TYPE "READ_AXES_POSITIONS_CH"
// stored: IsFailsafeCompliant false
   STRUCT
      READING_FAULT_1 : Bool;   // READING FAULT 1
      READING_DONE_1 : Bool;   // READING DONE 1
      REQUEST_1 : Bool;   // REQUEST 1
      READING_FAULT_2 : Bool;   // READING FAULT 2
      READING_DONE_2 : Bool;   // READING DONE 2
      REQUEST_2 : Bool;   // REQUEST 2
      READING_FAULT_3 : Bool;   // READING FAULT 3
      READING_DONE_3 : Bool;   // READING DONE 3
      REQUEST_3 : Bool;   // REQUEST 3
      FAULT_1 : Bool;   // FAULT 1
      FAULT_2 : Bool;   // FAULT 2
      FAULT_3 : Bool;   // FAULT 3
      IS : Bool;   // INMEDIATE STOP ALARMS / IMMEDIATE STOP ALARMS
      IS_SEOC : Bool;   // INMEDIATE STOP & STOP END OF CYCLE ALARMS / IMMEDIATE STOP & STOP END OF CYCLE ALARMS
      RHP : Bool;   // RETURN HOME POSITION ALARMS
      RHP_SEOC : Bool;   // RETURN HOME POSITION & STOP END OF CYCLE ALARMS
      SEOC : Bool;   // STOP END OF CYCLE ALARMS
      IS_WARNING : Bool;   // INMEDIATE STOP WARNING / IMMEDIATE STOP WARNING
      RHP_WARNING : Bool;   // RETURN HOME POSITION WARNING
      SEOC_WARNING : Bool;   // STOP END OF CYCLE WARNING
      WARNINGS : Bool;   // WARNINGS
      Help : Bool;   // Help
      Aux : Bool;   // Aux
      Aux1 : Bool;   // Aux1
      Aux2 : Bool;   // Aux2
      Aux3 : Bool;   // Aux3
      Aux4 : Bool;   // Aux4
      Aux5 : Bool;   // Aux5
      Aux6 : Bool;   // Aux6
      Aux7 : Bool;   // Aux7
      READING_STATUS : Word;   // READING STATUS
      POSITION_AXIS_1 : DWord;   // POSITION AXIS 1
      POSITION_AXIS_2 : DWord;   // POSITION AXIS 2
      POSITION_AXIS_3 : DWord;   // POSITION AXIS 3
      POSITION_AXIS_4 : DWord;   // POSITION AXIS 4
      POSITION_AXIS_5 : DWord;   // POSITION AXIS 5
      POSITION_AXIS_6 : DWord;   // POSITION AXIS 6
      POSITION_AXIS_7 : DWord;   // POSITION AXIS 7
      POSITION_AXIS_8 : DWord;   // POSITION AXIS 8
      POSITION_AXIS_9 : DWord;   // POSITION AXIS 9
      POSITION_AXIS_10 : DWord;   // POSITION AXIS 10
      POSITION_AXIS_11 : DWord;   // POSITION AXIS 11
      POSITION_AXIS_12 : DWord;   // POSITION AXIS 12
      POSITION_AXIS_13 : DWord;   // POSITION AXIS 13
      POSITION_AXIS_14 : DWord;   // POSITION AXIS 14
      POSITION_AXIS_15 : DWord;   // POSITION AXIS 15
      POSITION_AXIS_16 : DWord;   // POSITION AXIS 16
      POSITION_AXIS_17 : DWord;   // POSITION AXIS 17
      POSITION_AXIS_18 : DWord;   // POSITION AXIS 18
      POSITION_AXIS_19 : DWord;   // POSITION AXIS 19
      POSITION_AXIS_20 : DWord;   // POSITION AXIS 20
      CH_Reading_1 : Struct   // CH Reading 1
         SYNTAX_ID : Byte := BYTE#16#82;   // SYNTAX ID
         Area_Unit : Byte := BYTE#16#41;   // Area_Unit
         Column : Word := WORD#16#0002;   // Column
         Line : Word := WORD#16#0001;   // Line
         BlockType : Byte := BYTE#16#74;   // Block Type
         NumOfLine : Byte := BYTE#16#01;   // Number Of Line
         DataType : Byte := BYTE#16#0F;   // Data Type
         Length : Byte := BYTE#16#08;   // Length
      END_STRUCT;
      CH_Reading_2 : Struct   // CH Reading 2
         SYNTAX_ID : Byte := BYTE#16#82;   // SYNTAX ID
         Area_Unit : Byte := BYTE#16#41;   // Area_Unit
         Column : Word := WORD#16#0002;   // Column
         Line : Word := WORD#16#0002;   // Line
         BlockType : Byte := BYTE#16#74;   // Block Type
         NumOfLine : Byte := BYTE#16#01;   // Number Of Line
         DataType : Byte := BYTE#16#0F;   // Data Type
         Length : Byte := BYTE#16#08;   // Length
      END_STRUCT;
      CH_Reading_3 : Struct   // CH Reading 3
         SYNTAX_ID : Byte := BYTE#16#82;   // SYNTAX ID
         Area_Unit : Byte := BYTE#16#41;   // Area_Unit
         Column : Word := WORD#16#0002;   // Column
         Line : Word := WORD#16#0003;   // Line
         BlockType : Byte := BYTE#16#74;   // Block Type
         NumOfLine : Byte := BYTE#16#01;   // Number Of Line
         DataType : Byte := BYTE#16#0F;   // Data Type
         Length : Byte := BYTE#16#08;   // Length
      END_STRUCT;
      CH_Reading_4 : Struct   // CH Reading 4
         SYNTAX_ID : Byte := BYTE#16#82;   // SYNTAX ID
         Area_Unit : Byte := BYTE#16#41;   // Area_Unit
         Column : Word := WORD#16#0002;   // Column
         Line : Word := WORD#16#0004;   // Line
         BlockType : Byte := BYTE#16#74;   // Block Type
         NumOfLine : Byte := BYTE#16#01;   // Number Of Line
         DataType : Byte := BYTE#16#0F;   // Data Type
         Length : Byte := BYTE#16#08;   // Length
      END_STRUCT;
      CH_Reading_5 : Struct   // CH Reading 5
         SYNTAX_ID : Byte := BYTE#16#82;   // SYNTAX ID
         Area_Unit : Byte := BYTE#16#41;   // Area_Unit
         Column : Word := WORD#16#0002;   // Column
         Line : Word := WORD#16#0005;   // Line
         BlockType : Byte := BYTE#16#74;   // Block Type
         NumOfLine : Byte := BYTE#16#01;   // Number Of Line
         DataType : Byte := BYTE#16#0F;   // Data Type
         Length : Byte := BYTE#16#08;   // Length
      END_STRUCT;
      CH_Reading_6 : Struct   // CH Reading 6
         SYNTAX_ID : Byte := BYTE#16#82;   // SYNTAX ID
         Area_Unit : Byte := BYTE#16#41;   // Area_Unit
         Column : Word := WORD#16#0002;   // Column
         Line : Word := WORD#16#0006;   // Line
         BlockType : Byte := BYTE#16#74;   // Block Type
         NumOfLine : Byte := BYTE#16#01;   // Number Of Line
         DataType : Byte := BYTE#16#0F;   // Data Type
         Length : Byte := BYTE#16#08;   // Length
      END_STRUCT;
      CH_Reading_7 : Struct   // CH Reading 7
         SYNTAX_ID : Byte := BYTE#16#82;   // SYNTAX ID
         Area_Unit : Byte := BYTE#16#41;   // Area_Unit
         Column : Word := WORD#16#0002;   // Column
         Line : Word := WORD#16#0007;   // Line
         BlockType : Byte := BYTE#16#74;   // Block Type
         NumOfLine : Byte := BYTE#16#01;   // Number Of Line
         DataType : Byte := BYTE#16#0F;   // Data Type
         Length : Byte := BYTE#16#08;   // Length
      END_STRUCT;
      CH_Reading_8 : Struct   // CH Reading 8
         SYNTAX_ID : Byte := BYTE#16#82;   // SYNTAX ID
         Area_Unit : Byte := BYTE#16#41;   // Area_Unit
         Column : Word := WORD#16#0002;   // Column
         Line : Word := WORD#16#0008;   // Line
         BlockType : Byte := BYTE#16#74;   // Block Type
         NumOfLine : Byte := BYTE#16#01;   // Number Of Line
         DataType : Byte := BYTE#16#0F;   // Data Type
         Length : Byte := BYTE#16#08;   // Length
      END_STRUCT;
      CH_Reading_9 : Struct   // CH Reading 9
         SYNTAX_ID : Byte := BYTE#16#82;   // SYNTAX ID
         Area_Unit : Byte := BYTE#16#41;   // Area_Unit
         Column : Word := WORD#16#0002;   // Column
         Line : Word := WORD#16#0009;   // Line
         BlockType : Byte := BYTE#16#74;   // Block Type
         NumOfLine : Byte := BYTE#16#01;   // Number Of Line
         DataType : Byte := BYTE#16#0F;   // Data Type
         Length : Byte := BYTE#16#08;   // Length
      END_STRUCT;
      CH_Reading_10 : Struct   // CH Reading 10
         SYNTAX_ID : Byte := BYTE#16#82;   // SYNTAX ID
         Area_Unit : Byte := BYTE#16#41;   // Area_Unit
         Column : Word := WORD#16#0002;   // Column
         Line : Word := WORD#16#000A;   // Line
         BlockType : Byte := BYTE#16#73;   // Block Type
         NumOfLine : Byte := BYTE#16#01;   // Number Of Line
         DataType : Byte := BYTE#16#0F;   // Data Type
         Length : Byte := BYTE#16#08;   // Length
      END_STRUCT;
      CH_Reading_11 : Struct   // CH Reading 11
         SYNTAX_ID : Byte := BYTE#16#82;   // SYNTAX ID
         Area_Unit : Byte := BYTE#16#41;   // Area_Unit
         Column : Word := WORD#16#0002;   // Column
         Line : Word := WORD#16#000B;   // Line
         BlockType : Byte := BYTE#16#74;   // Block Type
         NumOfLine : Byte := BYTE#16#01;   // Number Of Line
         DataType : Byte := BYTE#16#0F;   // Data Type
         Length : Byte := BYTE#16#08;   // Length
      END_STRUCT;
      CH_Reading_12 : Struct   // CH Reading 12
         SYNTAX_ID : Byte := BYTE#16#82;   // SYNTAX ID
         Area_Unit : Byte := BYTE#16#41;   // Area_Unit
         Column : Word := WORD#16#0002;   // Column
         Line : Word := WORD#16#000C;   // Line
         BlockType : Byte := BYTE#16#74;   // Block Type
         NumOfLine : Byte := BYTE#16#01;   // Number Of Line
         DataType : Byte := BYTE#16#0F;   // Data Type
         Length : Byte := BYTE#16#08;   // Length
      END_STRUCT;
      CH_Reading_13 : Struct   // CH Reading 13
         SYNTAX_ID : Byte := BYTE#16#82;   // SYNTAX ID
         Area_Unit : Byte := BYTE#16#41;   // Area_Unit
         Column : Word := WORD#16#0002;   // Column
         Line : Word := WORD#16#000D;   // Line
         BlockType : Byte := BYTE#16#74;   // Block Type
         NumOfLine : Byte := BYTE#16#01;   // Number Of Line
         DataType : Byte := BYTE#16#0F;   // Data Type
         Length : Byte := BYTE#16#08;   // Length
      END_STRUCT;
      CH_Reading_14 : Struct   // CH Reading 14
         SYNTAX_ID : Byte := BYTE#16#82;   // SYNTAX ID
         Area_Unit : Byte := BYTE#16#41;   // Area_Unit
         Column : Word := WORD#16#0002;   // Column
         Line : Word := WORD#16#000E;   // Line
         BlockType : Byte := BYTE#16#74;   // Block Type
         NumOfLine : Byte := BYTE#16#01;   // Number Of Line
         DataType : Byte := BYTE#16#0F;   // Data Type
         Length : Byte := BYTE#16#08;   // Length
      END_STRUCT;
      CH_Reading_15 : Struct   // CH Reading 15
         SYNTAX_ID : Byte := BYTE#16#82;   // SYNTAX ID
         Area_Unit : Byte := BYTE#16#41;   // Area_Unit
         Column : Word := WORD#16#0002;   // Column
         Line : Word := WORD#16#000F;   // Line
         BlockType : Byte := BYTE#16#74;   // Block Type
         NumOfLine : Byte := BYTE#16#01;   // Number Of Line
         DataType : Byte := BYTE#16#0F;   // Data Type
         Length : Byte := BYTE#16#08;   // Length
      END_STRUCT;
      CH_Reading_16 : Struct   // CH Reading 16
         SYNTAX_ID : Byte := BYTE#16#82;   // SYNTAX ID
         Area_Unit : Byte := BYTE#16#41;   // Area_Unit
         Column : Word := WORD#16#0002;   // Column
         Line : Word := WORD#16#0010;   // Line
         BlockType : Byte := BYTE#16#74;   // Block Type
         NumOfLine : Byte := BYTE#16#01;   // Number Of Line
         DataType : Byte := BYTE#16#0F;   // Data Type
         Length : Byte := BYTE#16#08;   // Length
      END_STRUCT;
      CH_Reading_17 : Struct   // CH Reading 17
         SYNTAX_ID : Byte := BYTE#16#82;   // SYNTAX ID
         Area_Unit : Byte := BYTE#16#41;   // Area_Unit
         Column : Word := WORD#16#0002;   // Column
         Line : Word := WORD#16#0011;   // Line
         BlockType : Byte := BYTE#16#74;   // Block Type
         NumOfLine : Byte := BYTE#16#01;   // Number Of Line
         DataType : Byte := BYTE#16#0F;   // Data Type
         Length : Byte := BYTE#16#08;   // Length
      END_STRUCT;
      CH_Reading_18 : Struct   // CH Reading 18
         SYNTAX_ID : Byte := BYTE#16#82;   // SYNTAX ID
         Area_Unit : Byte := BYTE#16#41;   // Area_Unit
         Column : Word := WORD#16#0002;   // Column
         Line : Word := WORD#16#0012;   // Line
         BlockType : Byte := BYTE#16#74;   // Block Type
         NumOfLine : Byte := BYTE#16#01;   // Number Of Line
         DataType : Byte := BYTE#16#0F;   // Data Type
         Length : Byte := BYTE#16#08;   // Length
      END_STRUCT;
      CH_Reading_19 : Struct   // CH Reading 19
         SYNTAX_ID : Byte := BYTE#16#82;   // SYNTAX ID
         Area_Unit : Byte := BYTE#16#41;   // Area_Unit
         Column : Word := WORD#16#0002;   // Column
         Line : Word := WORD#16#0013;   // Line
         BlockType : Byte := BYTE#16#74;   // Block Type
         NumOfLine : Byte := BYTE#16#01;   // Number Of Line
         DataType : Byte := BYTE#16#0F;   // Data Type
         Length : Byte := BYTE#16#08;   // Length
      END_STRUCT;
      CH_Reading_20 : Struct   // CH Reading 20
         SYNTAX_ID : Byte := BYTE#16#82;   // SYNTAX ID
         Area_Unit : Byte := BYTE#16#41;   // Area_Unit
         Column : Word := WORD#16#0002;   // Column
         Line : Word := WORD#16#0014;   // Line
         BlockType : Byte := BYTE#16#74;   // Block Type
         NumOfLine : Byte := BYTE#16#01;   // Number Of Line
         DataType : Byte := BYTE#16#0F;   // Data Type
         Length : Byte := BYTE#16#08;   // Length
      END_STRUCT;
   END_STRUCT;
END_TYPE

TYPE "ASPIRATION"
// stored: IsFailsafeCompliant false
   STRUCT
      GENERAL_CONDITIONS : Bool;   // GENERAL CONDITIONS
      SWITCH_ON_CONDITIONS : Bool;   // ADVANCE CONDITIONS / SWITCH ON CONDITIONS
      SWITCH_OFF_CONDITIONS : Bool;   // RETURN CONDITIONS / SWITCH OFF CONDITIONS
      GENERAL_CONDITIONS_HELP : Bool;   // GENERAL CONDITIONS HELP
      SWITCH_ON_CONDITIONS_HELP : Bool;   // SWITCH ON CONDITIONS HELP
      SWITCH_OFF_CONDITIONS_HELP : Bool;   // SWITCH OFF CONDITIONS HELP
      SWITCH_ON_HMI_REQUEST : Bool;   // ADVANCE HMI REQUEST / SWITCH ON MANUAL HMI REQUEST
      SWITCH_OFF_HMI_REQUEST : Bool;   // RETURN HMI REQUEST / SWITCH OFF MANUAL HMI REQUEST
      SWITCH_ON_MANUAL_REQUEST : Bool;   // ADVANCE MANUAL REQUEST / SWITCH ON MANUAL REQUEST
      SWITCH_OFF_MANUAL_REQUEST : Bool;   // RETURN MANUAL REQUEST / SWITCH OFF MANUAL REQUEST
      SWITCH_ON_AUTO_REQUEST : Bool;   // ADVANCE AUTO REQUEST / SWITCH ON AUTO REQUEST
      SWITCH_OFF_AUTO_REQUEST : Bool;   // RETURN AUTO REQUEST / SWITCH OFF AUTO REQUEST
      SWITCH_ON_GLOBAL_REQUEST : Bool;   // ADVANCE GLOBAL REQUEST / SWITCH ON GLOBAL REQUEST
      SWITCH_OFF_GLOBAL_REQUEST : Bool;   // RETURN GLOBAL REQUEST / SWITCH OFF GLOBAL REQUEST
      SWITCH_ON_COMMAND : Bool;   // ADVANCE COMMAND / SWITCH ON COMMAND
      SWITCH_OFF_COMMAND : Bool;   // RETURN COMMAND / SWITCH OFF COMMAND
      FULL_SWITCHED_ON : Bool;   // ADVANCED FEEDBACK / SWITCHED ON AND COMMANDED
      FULL_SWITCHED_OFF : Bool;   // RETURNED FEEDBACK / SWITCHED OFF AND COMMANDED
      SIMULTANEITY_ALARM : Bool;   // SIMULTANEITY FAULT / SIMULTANEITY ALARM
      TIME_EXCEEDED_ALARM : Bool;   // TIME EXCEEDED / TIME EXCEEDED ALARM
      ANY_ACTIVE_ALARM : Bool;   // FAULT / ANY ACTIVE ALARM
      IS_SEOC_ALARMS : Bool;   // INMEDIATE STOP AND STOP END OF CYCLE ALARMS
      PULSE_1 : Bool;   // PULSE 1
      PULSE_2 : Bool;   // PULSE 2
      PULSE_3 : Bool;   // PULSE 3
   END_STRUCT;
END_TYPE

TYPE "CYL_ALARMS_OPN_CLS"
// stored: IsFailsafeCompliant false
   STRUCT
      CLOSED_SIMULTANEITY_1_ALARM : Bool;   // CLOSED SIMULTANEITY 1 ALARM
      CLOSED_TIME_EXCEEDED_1_ALARM : Bool;   // CLOSED TIME EXCEEDED 1 ALARM
      CLOSED_MISSING_1_ALARM : Bool;   // CLOSED MISSING 1 ALARM
      SPARE_1 : Bool;
      CLOSED_SIMULTANEITY_2_ALARM : Bool;   // CLOSED SIMULTANEITY 2 ALARM
      CLOSED_TIME_EXCEEDED_2_ALARM : Bool;   // CLOSED TIME EXCEEDED 2 ALARM
      CLOSED_MISSING_2_ALARM : Bool;   // CLOSED MISSING 2 ALARM
      SPARE_2 : Bool;
      CLOSED_SIMULTANEITY_3_ALARM : Bool;   // CLOSED SIMULTANEITY 3 ALARM
      CLOSED_TIME_EXCEEDED_3_ALARM : Bool;   // CLOSED TIME EXCEEDED 3 ALARM
      CLOSED_MISSING_3_ALARM : Bool;   // CLOSED MISSING 3 ALARM
      SPARE_3 : Bool;
      CLOSED_SIMULTANEITY_4_ALARM : Bool;   // CLOSED SIMULTANEITY 4 ALARM
      CLOSED_TIME_EXCEEDED_4_ALARM : Bool;   // CLOSED TIME EXCEEDED 4 ALARM
      CLOSED_MISSING_4_ALARM : Bool;   // CLOSED MISSING 4 ALARM
      SPARE_4 : Bool;
      CLOSED_OUTPUT_COMMAND_MISSING_ALARM : Bool;   // CLOSED OUTPUT COMMAND MISSING ALARM
      CLOSED_PRESSURE_TIME_EXCEEDED_1_ALARM : Bool;   // CLOSED PRESSURE TIME EXCEEDED 1 ALARM
      CLOSED_PRESSURE_SWITCH_1_ALARM : Bool;   // CLOSED PRESSURE SWITCH 1 ALARM
      CLOSED_PRESSURE_MISSING_1_ALARM : Bool;   // CLOSED PRESSURE MISSING 1 ALARM
      SPARE_5 : Bool;
      CLOSED_PRESSURE_TIME_EXCEEDED_2_ALARM : Bool;   // CLOSED PRESSURE TIME EXCEEDED 2 ALARM
      CLOSED_PRESSURE_SWITCH_2_ALARM : Bool;   // CLOSED PRESSURE SWITCH 2 ALARM
      CLOSED_PRESSURE_MISSING_2_ALARM : Bool;   // CLOSED PRESSURE MISSING 2 ALARM
      SPARE_6 : Bool;
      SPARE_7 : Bool;
      SPARE_8 : Bool;
      SPARE_9 : Bool;
      SPARE_10 : Bool;
      SPARE_11 : Bool;
      SPARE_12 : Bool;
      SPARE_13 : Bool;
      CLOSED_LOW_PRESSURE_TIME_EXCEEDED_ALARM : Bool;   // CLOSED LOW PRESSURE TIME EXCEEDED ALARM
      CLOSED_LOW_PRESSURE_SWITCH_ALARM : Bool;   // CLOSED LOW PRESSURE SWITCH ALARM
      CLOSED_LOW_PRESSURE_MISSING_ALARM : Bool;   // CLOSED LOW PRESSURE MISSING ALARM
      CLOSED_LOW_PRESSURE_OUTPUT_COMMAND_MISSING_ALARM : Bool;   // CLOSED LOW PRESSURE OUTPUT COMMAND MISSING ALARM
      SPARE_15 : Bool;
      SPARE_16 : Bool;
      SPARE_17 : Bool;
      SPARE_18 : Bool;
      OPEN_LOW_PRESSURE_TIME_EXCEEDED_ALARM : Bool;   // OPEN LOW PRESSURE TIME EXCEEDED ALARM
      OPEN_LOW_PRESSURE_SWITCH_ALARM : Bool;   // OPEN LOW PRESSURE SWITCH ALARM
      OPEN_LOW_PRESSURE_MISSING_ALARM : Bool;   // OPEN LOW PRESSURE MISSING ALARM
      OPEN_LOW_PRESSURE_OUTPUT_COMMAND_MISSING_ALARM : Bool;   // OPEN LOW PRESSURE OUTPUT COMMAND MISSING ALARM
      SPARE_23 : Bool;
      SPARE_24 : Bool;
      SPARE_25 : Bool;
      SPARE_26 : Bool;
      OPEN_SIMULTANEITY_1_ALARM : Bool;   // OPEN SIMULTANEITY 1 ALARM
      OPEN_TIME_EXCEEDED_1_ALARM : Bool;   // OPEN TIME EXCEEDED 1 ALARM
      OPEN_MISSING_1_ALARM : Bool;   // OPEN MISSING 1 ALARM
      SPARE_27 : Bool;
      OPEN_SIMULTANEITY_2_ALARM : Bool;   // OPEN SIMULTANEITY 2 ALARM
      OPEN_TIME_EXCEEDED_2_ALARM : Bool;   // OPEN TIME EXCEEDED 2 ALARM
      OPEN_MISSING_2_ALARM : Bool;   // OPEN MISSING 2 ALARM
      SPARE_28 : Bool;
      OPEN_SIMULTANEITY_3_ALARM : Bool;   // OPEN SIMULTANEITY 3 ALARM
      OPEN_TIME_EXCEEDED_3_ALARM : Bool;   // OPEN TIME EXCEEDED 3 ALARM
      OPEN_MISSING_3_ALARM : Bool;   // OPEN MISSING 3 ALARM
      SPARE_29 : Bool;
      OPEN_SIMULTANEITY_4_ALARM : Bool;   // OPEN SIMULTANEITY 4 ALARM
      OPEN_TIME_EXCEEDED_4_ALARM : Bool;   // OPEN TIME EXCEEDED 4 ALARM
      OPEN_MISSING_4_ALARM : Bool;   // OPEN MISSING 4 ALARM
      SPARE_30 : Bool;
      OPEN_OUTPUT_COMMAND_MISSING_ALARM : Bool;   // OPEN OUTPUT COMMAND MISSING ALARM
      OPEN_PRESSURE_TIME_EXCEEDED_1_ALARM : Bool;   // OPEN PRESSURE TIME EXCEEDED 1 ALARM
      OPEN_PRESSURE_SWITCH_1_ALARM : Bool;   // OPEN PRESSURE SWITCH 1 ALARM
      OPEN_PRESSURE_MISSING_1_ALARM : Bool;   // OPEN PRESSURE MISSING 1 ALARM
      SPARE_31 : Bool;
      OPEN_PRESSURE_TIME_EXCEEDED_2_ALARM : Bool;   // OPEN PRESSURE TIME EXCEEDED 2 ALARM
      OPEN_PRESSURE_SWITCH_2_ALARM : Bool;   // OPEN PRESSURE SWITCH 2 ALARM
      OPEN_PRESSURE_MISSING_2_ALARM : Bool;   // OPEN PRESSURE MISSING 2 ALARM
      SPARE_32 : Bool;
      SPARE_33 : Bool;
      SPARE_34 : Bool;
      SPARE_35 : Bool;
      SPARE_36 : Bool;
      SPARE_37 : Bool;
      SPARE_38 : Bool;
      SPARE_39 : Bool;
   END_STRUCT;
END_TYPE

TYPE "SMC_JXCP1_FROM_PLC"
// stored: IsFailsafeCompliant false
   STRUCT
      STEP_NUMBER_IN_0 : Bool := false;   // STEP NUMBER BINARY DIGIT 0
      STEP_NUMBER_IN_1 : Bool := false;   // STEP NUMBER BINARY DIGIT 1
      STEP_NUMBER_IN_2 : Bool := false;   // STEP NUMBER BINARY DIGIT 2
      STEP_NUMBER_IN_3 : Bool := false;   // STEP NUMBER BINARY DIGIT 3
      STEP_NUMBER_IN_4 : Bool := false;   // STEP NUMBER BINARY DIGIT 4
      STEP_NUMBER_IN_5 : Bool := false;   // STEP NUMBER BINARY DIGIT 5
      STEP_NUMBER_UNUSED_6 : Bool := false;   // -
      STEP_NUMBER_UNUSED_7 : Bool := false;   // -
      HOLD : Bool;   // HOLD - ACTUATOR STOP
      SVON : Bool;   // SERVO ON
      DRIVE : Bool;   // DRIVE ON
      RESET : Bool;   // RESET ALARM AND OPERATION
      SETUP : Bool;   // RETURN TO ORIGIN OPERATION
      JOG_MINUS : Bool;   // JOG MINUS DIRECTION
      JOG_PLUS : Bool;   // JOG PLUS DIRECTION
      FLGTH : Bool;   // INCHING FUNCTION
      UNUSED_2_0 : Bool;   // -
      SPEED_RESTRICTION : Bool;   // SPEED RESTRICTED
      UNUSED_2_2 : Bool;   // -
      UNUSED_2_3 : Bool;   // -
      MOVEMENT_MODE : Bool;   // MOVEMENT MODE
      SPEED_BIT : Bool;   // SPEED MODE
      POSITION : Bool;   // POSITION MODE
      ACCELERATION_BIT : Bool;   // ACELERATION MODE
      DECELERATION_BIT : Bool;   // DECELERATION MODE
      PUSHING_FORCE_BIT : Bool;   // PUSHING FORCE MODE
      TRIGGER_LV_BIT : Bool;   // TRIGGER LV MODE
      PUSHING_SPEED_BIT : Bool;   // PUSHING SPEED MODE
      MOVING_FORCE_BIT : Bool;   // MOVING FORCE MODE
      AREA_1_BIT : Bool;   // AREA 1
      AREA_2_BIT : Bool;   // AREA 2
      IN_POSITION_BIT : Bool;   // IN POSITION
      START_FLAG : Bool;   // TRANSMITING NUMERICAL INSTRUCTIONS
      UNUSED_4_1 : Bool;   // -
      UNUSED_4_2 : Bool;   // -
      UNUSED_4_3 : Bool;   // -
      UNUSED_4_4 : Bool;   // -
      UNUSED_4_5 : Bool;   // -
      UNUSED_4_6 : Bool;   // -
      UNUSED_4_7 : Bool;   // -
      MOVEMENT_MODE_BIT_0 : Bool;   // MOVEMENT BIT 0 --> 1:ABS(ABSOLUTE) / 2: INC(RELATIVE)
      MOVEMENT_MODE_BIT_1 : Bool;   // MOVEMENT BIT 1 --> 1:ABS(ABSOLUTE) / 2: INC(RELATIVE)
      UNUSED_5_2 : Bool;   // -
      UNUSED_5_3 : Bool;   // -
      UNUSED_5_4 : Bool;   // -
      UNUSED_5_5 : Bool;   // -
      UNUSED_5_6 : Bool;   // -
      UNUSED_5_7 : Bool;   // -
      SPEED_VALUE : Word;   // SPEED VALUE (1mm/s)
      TARGET_POSITION : DWord;   // TARGET POSITION (0.01mm)
      ACCELERATION_VALUE : Word;   // ACCELERATION VALUE (1mm/s2)
      DECELERATION_VALUE : Word;   // DECELERATION VALUE (1mm/s2)
      PUSHING_FORCE_VALUE : Word;   // PUSHING FORCE VALUE (%)
      TRIGGER_LV_VALUE : Word;   // TRIGGER LV VALUE (%)
      PUSHING_SPEED_VALUE : Word;   // PUSHING SPEED VALEU (1mm/s)
      MOVING_FORCE_VALUE : Word;   // MOVING FORCE VALUE (%)
      AREA_1_VALUE : Word;   // AREA 1 VALUE (0.01mm)
      AREA_2_VALUE : Word;   // AREA 2 VALUE (0.01mm)
      IN_POSITION_VALUE : Word;   // IN POSITION VALUE (0.01mm)
   END_STRUCT;
END_TYPE

TYPE "SMC_JXCP1_TO_PLC"
// stored: IsFailsafeCompliant false
   STRUCT
      STEP_NUMBER_OUT_0 : Bool := false;   // STEP NUMBER BINARY DIGIT 0
      STEP_NUMBER_OUT_1 : Bool := false;   // STEP NUMBER BINARY DIGIT 1
      STEP_NUMBER_OUT_2 : Bool := false;   // STEP NUMBER BINARY DIGIT 2
      STEP_NUMBER_OUT_3 : Bool := false;   // STEP NUMBER BINARY DIGIT 3
      STEP_NUMBER_OUT_4 : Bool := false;   // STEP NUMBER BINARY DIGIT 4
      STEP_NUMBER_OUT_5 : Bool := false;   // STEP NUMBER BINARY DIGIT 5
      STEP_NUMBER_UNUSED_6 : Bool := false;   // -
      STEP_NUMBER_UNUSED_7 : Bool := false;   // -
      BUSY : Bool;   // CONTROLLER BUSY (MOVEMENT)
      SVRE : Bool;   // SERVO MOTOR STATUS (ON/OFF)
      STON : Bool;   // POSITION INFORMATION/STATUS ESTABLISHED
      INP : Bool;   // IN POSITION
      AREA : Bool;   // BETWEEN AREA 1 AND AREA 2 IN STEP DATA
      WAREA : Bool;   // BETWEEN W AREA 1 AND W AREA 2 IN STEP DATA
      ESTOP : Bool;   // TEACHING BOX EMERGENCY STOP
      ALARM : Bool;   // ALARM PRESENT
      UNUSED_2_0 : Bool;   // -
      UNUSED_2_1 : Bool;   // -
      UNUSED_2_2 : Bool;   // -
      UNUSED_2_3 : Bool;   // -
      READY : Bool;   // SERVO ON AND NO ALARMS
      UNUSED_2_5 : Bool;   // -
      UNUSED_2_6 : Bool;   // -
      UNUSED_2_7 : Bool;   // -
      UNSUSED_3_0 : Bool;   // -
      UNSUSED_3_1 : Bool;   // -
      UNSUSED_3_2 : Bool;   // -
      UNSUSED_3_3 : Bool;   // -
      UNSUSED_3_4 : Bool;   // -
      UNSUSED_3_5 : Bool;   // -
      UNSUSED_3_6 : Bool;   // -
      UNSUSED_3_7 : Bool;   // -
      CURRENT_POSITION : DWord;   // CURRENT ACTUATOR POSITION (MULTIPLES OF 0.01mm)
      CURRENT_SPEED : Word;   // CURRENT ACTUATOR SPEED (MULTIPLES OF 1mm/s)
      CURRENT_PUSHING_FORCE : Word;   // CURRENT ACTUATOR PUSHING FORCE (MULTIPLES OF 1%)
      TARGET_POSITION : DWord;   // TARGET ACTUATOR POSITION (MULTIPLES OF 0.01mm)
      ALARM_1 : DWord;   // ALARM 1 CODE
      ALARM_2 : DWord;   // ALARM 2 CODE
      ALARM_3 : DWord;   // ALARM 3 CODE
      ALARM_4 : DWord;   // ALARM 4 CODE
   END_STRUCT;
END_TYPE

TYPE "CHANNEL_PLC_SIGNALS"
// stored: IsFailsafeCompliant false
   STRUCT
      INPUT : Struct
         START_POSITION_SIGNAL : Bool;
         RETURN_HOME_SIGNAL : Bool;
         START_TORQUE_SIGNAL : Bool;
      END_STRUCT;
      OUTPUT : Struct
         IN_POSITION_SIGNAL : Bool;
         IN_HOME_SIGNAL : Bool;
         IN_TORQUE_SIGNAL : Bool;
      END_STRUCT;
   END_STRUCT;
END_TYPE

TYPE "MR_J4_Aux_Control"
// stored: IsFailsafeCompliant false
   STRUCT
      Aux_Input : Struct
         SVON : Bool;
         SETUP : Bool;
         Jog_P : Bool;
         Jog_N : Bool;
         Reset : Bool;
         Hold : Bool;
         FLGTH : Bool;
         Speed_Restr : Bool;
         Start_Flag : Bool;
         Fly_Change : Bool;
         Continuous_Step : Bool;
      END_STRUCT;
      Aux_Output : Struct
         Svre : Bool;
         Seton : Bool;
         Busy : Bool;
         Inp : Bool;
         TLO : Bool;
         New_step_Ack : Bool;
         ILA : Bool;
         Warning : Bool;
         Alarm : Bool;
         Alarm_Bateria : Bool;
         Alarm_S_ABS : Bool;
         Voltage_Enable : Bool;
         LSN : Bool;
         LSP : Bool;
         Dog : Bool;
         STO1 : Bool;
         STO2 : Bool;
         Step_Actual : UInt;
         Pos_actual : DInt;
         Speed_Actual : Int;
         Par_Actual : Int;
         Pos_Pedida : DInt;
         Modo_Trabajo : Byte := 0;
         Alarma_Actual : DWord;
         Temperature_Encoder : DInt;
         Bus_Voltage : DInt;
         Efective_load_Ratio : DInt;
         Regenerative_load_Ratio : DInt;
      END_STRUCT;
      Aux_Param_Config : Struct
         Paso_Vuelta : UInt;
         "Velocidad maxima" : Int;
         Ac_DC_maxima : Int;
         Jog_speed : UInt;
         Jog_AC_DC : UInt;
         Torque_max_speed : Int;
         Torque_Max_TQ : Int;
         Torque_SLope_TQ : Int;
      END_STRUCT;
   END_STRUCT;
END_TYPE

TYPE "MR_J4_Step"
// stored: IsFailsafeCompliant false
   STRUCT
      Output : Struct
         Op_mode : Int;
         Speed : Int;
         Position : DInt;
         Acceleration : Int;
         Deceleration : Int;
         Pushing_Force : Int;
         Trigger_Level : Int;
         Pushing_Speed : Int;
         Inpos : DInt;
      END_STRUCT;
   END_STRUCT;
END_TYPE

TYPE "MR_J4_TN_Input"
// stored: IsFailsafeCompliant false
   STRUCT
      Input : Struct
         "I_mode operation_B1" : Byte;
         "I_mode operation_B2" : Byte;
         I_SW_B8 : Bool;
         I_SW_B9_RM : Bool;
         I_SW_B10_TR : Bool;
         I_SW_B11_ILA : Bool;
         I_SW_B12_SPoint : Bool;
         I_SW_B13_FError : Bool;
         I_SW_B14 : Bool;
         I_SW_B15 : Bool;
         I_SW_B0_RTSO : Bool;
         I_SW_B1_SO : Bool;
         I_SW_B2_0E : Bool;
         I_SW_B3_Fault : Bool;
         I_SW_B4_VE : Bool;
         I_SW_B5_QS : Bool;
         I_SW_B6_SOD : Bool;
         I_SW_B7_Warning : Bool;
         I_SDO1_B8 : Bool;
         I_SDO1_B9 : Bool;
         I_SDO1_B10 : Bool;
         I_SDO1_B11 : Bool;
         I_SDO1_B12_S_INP : Bool;
         I_SDO1_B13_S_TLC : Bool;
         I_SDO1_B14_S_ABSV : Bool;
         I_SDO1_B15_S_BWNG : Bool;
         I_SDO1_B0 : Bool;
         I_SDO1_B1 : Bool;
         I_SDO1_B2_S_SA : Bool;
         I_SDO1_B3_S_MBR : Bool;
         I_SDO1_B4_S_CDPS : Bool;
         I_SDO1_B5_S_CLD : Bool;
         I_SDO1_B6 : Bool;
         I_SDO1_B7 : Bool;
         I_SDO2_B8_S_PC : Bool;
         I_SDO2_B9 : Bool;
         I_SDO2_B10_S_DB : Bool;
         I_SDO2_B11 : Bool;
         I_SDO2_B12 : Bool;
         I_SDO2_B13 : Bool;
         I_SDO2_B14 : Bool;
         I_SDO2_B15_S_ZP2 : Bool;
         I_SDO2_B0_S_ZPAS : Bool;
         I_SDO2_B1 : Bool;
         I_SDO2_B2 : Bool;
         I_SDO2_B3_S_ZSP : Bool;
         I_SDO2_B4_S_VLC : Bool;
         I_SDO2_B5 : Bool;
         I_SDO2_B6_S_IPF : Bool;
         I_SDO2_B7 : Bool;
         I_SDO3 : Word;
         "I_Torque actual" : Int;
         "I_Digital input" : DWord;
         "I_Posicion actual" : DInt;
         "I_Velocity actual" : DInt;
         "I_Following error" : DInt;
         "I_Touch probe_pos1 pos" : DInt;
         "I_Touch_probe_pos1 neg" : DInt;
         "I_Touch_probe_pos2 pos" : DInt;
         "I_Touch_probe_pos2 neg" { ExternalAccessible := 'False'; ExternalVisible := 'False'; ExternalWritable := 'False'} : DInt;
         I_Touch_probe_status : Int;
         I_reserved : Word;
      END_STRUCT;
   END_STRUCT;
END_TYPE

TYPE "MR_J4_TN_Output"
// stored: IsFailsafeCompliant false
   STRUCT
      Output : Struct
         "Q_Mode opeation_B1" : Byte;
         "Q_Mode opeation_B2" : Byte;
         Q_CW_B8_Halt : Bool;
         Q_CW_B9_ChangeP2 : Bool;
         Q_CW_B10 : Bool;
         Q_CW_B11 : Bool;
         Q_CW_B12 : Bool;
         Q_CW_B13 : Bool;
         Q_CW_B14 : Bool;
         Q_CW_B15 : Bool;
         Q_CW_B0_SO : Bool;
         Q_CW_B1_EV : Bool;
         Q_CW_B2_QS : Bool;
         Q_CW_B3_EO : Bool;
         Q_CW_B4_Npoint : Bool;
         Q_CW_B5_ChangeP : Bool;
         Q_CW_B6_Abs_Rel : Bool;
         Q_CW_B7_FReset : Bool;
         "Q_Control DI 1" : Word;
         "Q_Control D12" : Word;
         "Q_Control DI 3" : Word;
         "Q_Target torque" : Int;
         "Q_Torque Slope" : DInt;
         "Q_Target position" : DInt;
         "Q_Taget velocity" : DInt;
         "Q_Velocity limit" : DInt;
         "Q_Profile velocity" : DInt;
         "Q_Profile acceleration" : DInt;
         "Q_Profile deeleration" : DInt;
         "Q_Touch probe" : Word;
         Q_reserved1 : Word;
         Q_reserved2 : Word;
         Q_reserved3 : Word;
      END_STRUCT;
   END_STRUCT;
END_TYPE

TYPE "MR_J4_TN_RDasincro"
// stored: IsFailsafeCompliant false
   STRUCT
      Id_Driver : HW_IO;
      Param_to_Read : DInt;
      Param_M_Len : UInt;
      Param_Value : Array[0..3] of Word;
      Len_InfoOut : UInt;
      Error_to_Read : UInt;
      Status_diagnosis : DWord;
   END_STRUCT;
END_TYPE

TYPE "U01_STA3_MEAS.U01_STA3_MEAS_Method.TriggerCalculateDistance.Inputs"
// stored: IsFailsafeCompliant false
   STRUCT
      DMC { ExternalAccessible := 'False'; ExternalVisible := 'False'; ExternalWritable := 'False'} : WString;
      "Fixture ID" { ExternalAccessible := 'False'; ExternalVisible := 'False'; ExternalWritable := 'False'} : Int;
   END_STRUCT;
END_TYPE

TYPE "U01_STA3_MEAS.U01_STA3_MEAS_Method.TriggerCalculateDistance.Outputs"
// stored: IsFailsafeCompliant false
   STRUCT
      Result { ExternalAccessible := 'False'; ExternalVisible := 'False'; ExternalWritable := 'False'} : Bool;
   END_STRUCT;
END_TYPE

TYPE "U01_STA3_MEAS.U01_STA3_MEAS_Method.TriggerCalibration.Inputs"
// stored: IsFailsafeCompliant false
   STRUCT
      "Fixture ID" { ExternalAccessible := 'False'; ExternalVisible := 'False'; ExternalWritable := 'False'} : Int;
   END_STRUCT;
END_TYPE

TYPE "U01_STA3_MEAS.U01_STA3_MEAS_Method.TriggerCalibration.Outputs"
// stored: IsFailsafeCompliant false
   STRUCT
      Result { ExternalAccessible := 'False'; ExternalVisible := 'False'; ExternalWritable := 'False'} : Bool;
   END_STRUCT;
END_TYPE

TYPE "U01_STA3_MEAS.U01_STA3_MEAS_Method.TriggerReset.Outputs"
// stored: IsFailsafeCompliant false
   STRUCT
      Result { ExternalAccessible := 'False'; ExternalVisible := 'False'; ExternalWritable := 'False'} : Bool;
   END_STRUCT;
END_TYPE

TYPE "U01_STA3_MEAS.U01_STA3_MEAS_Method.TriggerStartLayerThicknessAcquisition.Inputs"
// stored: IsFailsafeCompliant false
   STRUCT
      DMC { ExternalAccessible := 'False'; ExternalVisible := 'False'; ExternalWritable := 'False'} : WString;
      "Fixture ID" { ExternalAccessible := 'False'; ExternalVisible := 'False'; ExternalWritable := 'False'} : Int;
   END_STRUCT;
END_TYPE

TYPE "U01_STA3_MEAS.U01_STA3_MEAS_Method.TriggerStartLayerThicknessAcquisition.Outputs"
// stored: IsFailsafeCompliant false
   STRUCT
      Result { ExternalAccessible := 'False'; ExternalVisible := 'False'; ExternalWritable := 'False'} : Bool;
   END_STRUCT;
END_TYPE

TYPE "U01_STA3_MEAS.U01_STA3_MEAS_Method.TriggerStopLayerThicknessAcquisition.Outputs"
// stored: IsFailsafeCompliant false
   STRUCT
      Result { ExternalAccessible := 'False'; ExternalVisible := 'False'; ExternalWritable := 'False'} : Bool;
   END_STRUCT;
END_TYPE

TYPE "U01_STA3_MEAS.U01_STA3_MEAS_Read"
// stored: IsFailsafeCompliant false
   STRUCT
      Status { ExternalWritable := 'False'} : Int;
      ProfilerConfiguration { ExternalWritable := 'False'} : Bool;
      AnalyzerConfiguration { ExternalWritable := 'False'} : Bool;
      DMCStructure { ExternalWritable := 'False'} : Bool;
      Acquisition { ExternalWritable := 'False'} : Bool;
      ProfilerInitialization { ExternalWritable := 'False'} : Bool;
      DistanceCalculation { ExternalWritable := 'False'} : Bool;
      LayerThicknessAnalysis { ExternalWritable := 'False'} : Bool;
      StorageError { ExternalWritable := 'False'} : Bool;
      DatabaseConnection { ExternalWritable := 'False'} : Bool;
      SensorTemperature { ExternalWritable := 'False'} : Real;
      DistanceSurfaceToReference { ExternalWritable := 'False'} : Real;
      "Status Fixture 1" { ExternalWritable := 'False'} : Bool;
      "Status Fixture 2" { ExternalWritable := 'False'} : Bool;
      "Status Fixture 3" { ExternalWritable := 'False'} : Bool;
      "Status Fixture 4" { ExternalWritable := 'False'} : Bool;
   END_STRUCT;
END_TYPE

TYPE "U02_STA2_MEAS.U02_STA2_MEAS_Method.TriggerAnalysis.Inputs"
// stored: IsFailsafeCompliant false
   STRUCT
      DMC { ExternalAccessible := 'False'; ExternalVisible := 'False'; ExternalWritable := 'False'} : WString;
      "Fixture ID" { ExternalAccessible := 'False'; ExternalVisible := 'False'; ExternalWritable := 'False'} : Int;
   END_STRUCT;
END_TYPE

TYPE "U02_STA2_MEAS.U02_STA2_MEAS_Method.TriggerAnalysis.Outputs"
// stored: IsFailsafeCompliant false
   STRUCT
      Result { ExternalAccessible := 'False'; ExternalVisible := 'False'; ExternalWritable := 'False'} : Bool;
   END_STRUCT;
END_TYPE

TYPE "U02_STA2_MEAS.U02_STA2_MEAS_Method.TriggerCalibration.Inputs"
// stored: IsFailsafeCompliant false
   STRUCT
      "Fixture ID" { ExternalAccessible := 'False'; ExternalVisible := 'False'; ExternalWritable := 'False'} : Int;
   END_STRUCT;
END_TYPE

TYPE "U02_STA2_MEAS.U02_STA2_MEAS_Method.TriggerCalibration.Outputs"
// stored: IsFailsafeCompliant false
   STRUCT
      Result { ExternalAccessible := 'False'; ExternalVisible := 'False'; ExternalWritable := 'False'} : Bool;
   END_STRUCT;
END_TYPE

TYPE "U02_STA2_MEAS.U02_STA2_MEAS_Method.TriggerReset.Outputs"
// stored: IsFailsafeCompliant false
   STRUCT
      Result { ExternalAccessible := 'False'; ExternalVisible := 'False'; ExternalWritable := 'False'} : Bool;
   END_STRUCT;
END_TYPE

TYPE "U02_STA2_MEAS.U02_STA2_MEAS_Read"
// stored: IsFailsafeCompliant false
   STRUCT
      Status { ExternalWritable := 'False'} : Int;
      ProfilerConfiguration { ExternalWritable := 'False'} : Bool;
      AnalyzerConfiguration { ExternalWritable := 'False'} : Bool;
      DMCStructure { ExternalWritable := 'False'} : Bool;
      Acquisition { ExternalWritable := 'False'} : Bool;
      ProfilerInitialization { ExternalWritable := 'False'} : Bool;
      UmbrellaAnalysis { ExternalWritable := 'False'} : Bool;
      RunOutAnalysis { ExternalWritable := 'False'} : Bool;
      SurfaceDefectsAnalysis { ExternalWritable := 'False'} : Bool;
      StorageError { ExternalWritable := 'False'} : Bool;
      DatabaseConnection { ExternalWritable := 'False'} : Bool;
      SensorTemperature { ExternalWritable := 'False'} : Real;
      "Status Fixture 1" { ExternalWritable := 'False'} : Bool;
      "Status Fixture 2" { ExternalWritable := 'False'} : Bool;
      "Status Fixture 3" { ExternalWritable := 'False'} : Bool;
      "Status Fixture 4" { ExternalWritable := 'False'} : Bool;
   END_STRUCT;
END_TYPE

TYPE "U02_STA3_MEAS.U02_STA3_MEAS_Method.TriggerCalculateDistance.Inputs"
// stored: IsFailsafeCompliant false
   STRUCT
      DMC { ExternalAccessible := 'False'; ExternalVisible := 'False'; ExternalWritable := 'False'} : WString;
      "Fixture ID" { ExternalAccessible := 'False'; ExternalVisible := 'False'; ExternalWritable := 'False'} : Int;
   END_STRUCT;
END_TYPE

TYPE "U02_STA3_MEAS.U02_STA3_MEAS_Method.TriggerCalculateDistance.Outputs"
// stored: IsFailsafeCompliant false
   STRUCT
      Result { ExternalAccessible := 'False'; ExternalVisible := 'False'; ExternalWritable := 'False'} : Bool;
   END_STRUCT;
END_TYPE

TYPE "U02_STA3_MEAS.U02_STA3_MEAS_Method.TriggerCalibration.Inputs"
// stored: IsFailsafeCompliant false
   STRUCT
      "Fixture ID" { ExternalAccessible := 'False'; ExternalVisible := 'False'; ExternalWritable := 'False'} : Int;
   END_STRUCT;
END_TYPE

TYPE "U02_STA3_MEAS.U02_STA3_MEAS_Method.TriggerCalibration.Outputs"
// stored: IsFailsafeCompliant false
   STRUCT
      Result { ExternalAccessible := 'False'; ExternalVisible := 'False'; ExternalWritable := 'False'} : Bool;
   END_STRUCT;
END_TYPE

TYPE "U02_STA3_MEAS.U02_STA3_MEAS_Method.TriggerReset.Outputs"
// stored: IsFailsafeCompliant false
   STRUCT
      Result { ExternalAccessible := 'False'; ExternalVisible := 'False'; ExternalWritable := 'False'} : Bool;
   END_STRUCT;
END_TYPE

TYPE "U02_STA3_MEAS.U02_STA3_MEAS_Method.TriggerStartLayerThicknessAcquisition.Inputs"
// stored: IsFailsafeCompliant false
   STRUCT
      DMC { ExternalAccessible := 'False'; ExternalVisible := 'False'; ExternalWritable := 'False'} : WString;
      "Fixture ID" { ExternalAccessible := 'False'; ExternalVisible := 'False'; ExternalWritable := 'False'} : Int;
   END_STRUCT;
END_TYPE

TYPE "U02_STA3_MEAS.U02_STA3_MEAS_Method.TriggerStartLayerThicknessAcquisition.Outputs"
// stored: IsFailsafeCompliant false
   STRUCT
      Result { ExternalAccessible := 'False'; ExternalVisible := 'False'; ExternalWritable := 'False'} : Bool;
   END_STRUCT;
END_TYPE

TYPE "U02_STA3_MEAS.U02_STA3_MEAS_Method.TriggerStopLayerThicknessAcquisition.Outputs"
// stored: IsFailsafeCompliant false
   STRUCT
      Result { ExternalAccessible := 'False'; ExternalVisible := 'False'; ExternalWritable := 'False'} : Bool;
   END_STRUCT;
END_TYPE

TYPE "U02_STA3_MEAS.U02_STA3_MEAS_Read"
// stored: IsFailsafeCompliant false
   STRUCT
      Status { ExternalWritable := 'False'} : Int;
      ProfilerConfiguration { ExternalWritable := 'False'} : Bool;
      AnalyzerConfiguration { ExternalWritable := 'False'} : Bool;
      DMCStructure { ExternalWritable := 'False'} : Bool;
      Acquisition { ExternalWritable := 'False'} : Bool;
      ProfilerInitialization { ExternalWritable := 'False'} : Bool;
      DistanceCalculation { ExternalWritable := 'False'} : Bool;
      LayerThicknessAnalysis { ExternalWritable := 'False'} : Bool;
      StorageError { ExternalWritable := 'False'} : Bool;
      DatabaseConnection { ExternalWritable := 'False'} : Bool;
      SensorTemperature { ExternalWritable := 'False'} : Real;
      DistanceSurfaceToReference { ExternalWritable := 'False'} : Real;
      "Status Fixture 1" { ExternalWritable := 'False'} : Bool;
      "Status Fixture 2" { ExternalWritable := 'False'} : Bool;
      "Status Fixture 3" { ExternalWritable := 'False'} : Bool;
      "Status Fixture 4" { ExternalWritable := 'False'} : Bool;
   END_STRUCT;
END_TYPE

TYPE "U03_MEAS_STATION_FACE_A.U03_FACE_A_MEAS_Method.TriggerAnalysis.Inputs"
// stored: IsFailsafeCompliant false
   STRUCT
      DMC { ExternalAccessible := 'False'; ExternalVisible := 'False'; ExternalWritable := 'False'} : WString;
   END_STRUCT;
END_TYPE

TYPE "U03_MEAS_STATION_FACE_A.U03_FACE_A_MEAS_Method.TriggerAnalysis.Outputs"
// stored: IsFailsafeCompliant false
   STRUCT
      Result { ExternalAccessible := 'False'; ExternalVisible := 'False'; ExternalWritable := 'False'} : Bool;
   END_STRUCT;
END_TYPE

TYPE "U03_MEAS_STATION_FACE_A.U03_FACE_A_MEAS_Method.TriggerCalibration.Outputs"
// stored: IsFailsafeCompliant false
   STRUCT
      Result { ExternalAccessible := 'False'; ExternalVisible := 'False'; ExternalWritable := 'False'} : Bool;
   END_STRUCT;
END_TYPE

TYPE "U03_MEAS_STATION_FACE_A.U03_FACE_A_MEAS_Method.TriggerReset.Outputs"
// stored: IsFailsafeCompliant false
   STRUCT
      Result { ExternalAccessible := 'False'; ExternalVisible := 'False'; ExternalWritable := 'False'} : Bool;
   END_STRUCT;
END_TYPE

TYPE "U03_MEAS_STATION_FACE_A.U03_FACE_A_MEAS_Read"
// stored: IsFailsafeCompliant false
   STRUCT
      Status { ExternalWritable := 'False'} : Int;
      ProfilerConfiguration { ExternalWritable := 'False'} : Bool;
      AnalyzerConfiguration { ExternalWritable := 'False'} : Bool;
      DMCStructure { ExternalWritable := 'False'} : Bool;
      Acquisition { ExternalWritable := 'False'} : Bool;
      ProfilerInitialization { ExternalWritable := 'False'} : Bool;
      UmbrellaAnalysis { ExternalWritable := 'False'} : Bool;
      RunOutAnalysis { ExternalWritable := 'False'} : Bool;
      DistanceCalculation { ExternalWritable := 'False'} : Bool;
      SurfaceDefectsAnalysis { ExternalWritable := 'False'} : Bool;
      StorageError { ExternalWritable := 'False'} : Bool;
      DatabaseConnection { ExternalWritable := 'False'} : Bool;
      SensorTemperature { ExternalWritable := 'False'} : Real;
      "Status Fixture 1" { ExternalWritable := 'False'} : Bool;
   END_STRUCT;
END_TYPE

TYPE "U03_MEAS_STATION_FACE_B.U03_FACE_B_MEAS_Method.TriggerAnalysis.Inputs"
// stored: IsFailsafeCompliant false
   STRUCT
      DMC { ExternalAccessible := 'False'; ExternalVisible := 'False'; ExternalWritable := 'False'} : WString;
   END_STRUCT;
END_TYPE

TYPE "U03_MEAS_STATION_FACE_B.U03_FACE_B_MEAS_Method.TriggerAnalysis.Outputs"
// stored: IsFailsafeCompliant false
   STRUCT
      Result { ExternalAccessible := 'False'; ExternalVisible := 'False'; ExternalWritable := 'False'} : Bool;
   END_STRUCT;
END_TYPE

TYPE "U03_MEAS_STATION_FACE_B.U03_FACE_B_MEAS_Method.TriggerCalibration.Outputs"
// stored: IsFailsafeCompliant false
   STRUCT
      Result { ExternalAccessible := 'False'; ExternalVisible := 'False'; ExternalWritable := 'False'} : Bool;
   END_STRUCT;
END_TYPE

TYPE "U03_MEAS_STATION_FACE_B.U03_FACE_B_MEAS_Method.TriggerReset.Outputs"
// stored: IsFailsafeCompliant false
   STRUCT
      Result { ExternalAccessible := 'False'; ExternalVisible := 'False'; ExternalWritable := 'False'} : Bool;
   END_STRUCT;
END_TYPE

TYPE "U03_MEAS_STATION_FACE_B.U03_FACE_B_MEAS_Read"
// stored: IsFailsafeCompliant false
   STRUCT
      Status { ExternalWritable := 'False'} : Int;
      ProfilerConfiguration { ExternalWritable := 'False'} : Bool;
      AnalyzerConfiguration { ExternalWritable := 'False'} : Bool;
      DMCStructure { ExternalWritable := 'False'} : Bool;
      Acquisition { ExternalWritable := 'False'} : Bool;
      ProfilerInitialization { ExternalWritable := 'False'} : Bool;
      UmbrellaAnalysis { ExternalWritable := 'False'} : Bool;
      RunOutAnalysis { ExternalWritable := 'False'} : Bool;
      DistanceCalculation { ExternalWritable := 'False'} : Bool;
      SurfaceDefectsAnalysis { ExternalWritable := 'False'} : Bool;
      StorageError { ExternalWritable := 'False'} : Bool;
      DatabaseConnection { ExternalWritable := 'False'} : Bool;
      SensorTemperature { ExternalWritable := 'False'} : Real;
      "Status Fixture 1" { ExternalWritable := 'False'} : Bool;
   END_STRUCT;
END_TYPE

TYPE "LASER TRUMPF"
// stored: IsFailsafeCompliant false
   STRUCT
      OUTPUTS : Struct
         CONTROL : Struct
            LASER_REQUEST : Bool := FALSE;   // REQUESTING THE LASER
            PILOT_LASER_ON : Bool := FALSE;   // SWITCHING ON THE PILOT LASER
            UNSYNC_PSTART : Bool := FALSE;   // UNSYNCHRONIZED ACTIVATION
            SIMULATION : Bool := FALSE;   // SIMULATION MODE
            LOCK_PROG_PARAM : Bool := FALSE;   // ONLY FOR TRUMICRO: LOCK OPERATING POINT PARAMETERS. RESERVED FOR ALL OTHER LASER DEVICES.
            INQUIRY_2 : Bool := FALSE;   // QUERY INPUT 2
            INQUIRY_1 : Bool := FALSE;   // QUERY INPUT 1
            FAULT_EXTERNAL : Bool := FALSE;   // EXTERNAL FAULT
            RESET : Bool := FALSE;   // RESET
            PROGRAM_STOP : Bool := FALSE;   // CANCEL / STOP LASER PROGRAM
            PROG_START_DYN : Bool := FALSE;   // DYNAMIC PROGRAM START
            PROG_START_SATICAL : Bool := FALSE;   // STATIC PROGRAM START
            LASER_STANDBY : Bool := FALSE;   // ACTIVATING THE LASER STANDBY MODE
            LASER_ON : Bool := FALSE;   // SWITCHING ON THE LASER
            LOCK_OPERAT_PANEL : Bool := FALSE;   // LOCKING THE OPERATING PANE
            EXT_CONTROL : Bool := FALSE;   // EXTERNAL CONTROL
         END_STRUCT;
         PROGRAMNO : Byte := B#16#0;   // NUMBER OF THE SELECTED LASER PROGRAM
         LIGHTPATH : Byte := B#16#0;   // NUMBER OF THE SELECTED LIGHT PATH
         LASER_NO : Byte := B#16#0;   // NUMBER OF THE SELECTED LASER DEVICE
         AD_NO : Byte := B#16#0;   // NUMBER OF THE APPLICATION DATA SET
         POWER_VALUE : Word := W#16#0;   // POWER VALUE (IW3)
         PROCESSING : Word := W#16#0;   // PROCESSING (IW4)
         POWER_PORTION_CORE : Word;   // POWER PORTION CORE (IW5)
      END_STRUCT;
      INPUTS : Struct
         STATUS : Struct
            LASER_WARNING_LAP_ON : Bool := FALSE;   // THE LASER WARNING LIGHT IS ON
            PILOT_LASER_IS_ON : Bool := FALSE;   // PILOT LASER IS SWITCHED ON
            POWER_LIMIT : Bool := FALSE;   // THE POWER LIMIT OF THE LASER HAS BEEN REACHED
            LASER_ASSIGNED : Bool := FALSE;   // THE LASER DEVICE IS ASSIGNED TO AN EXTERNAL CONTROL UNIT
            FAULT_LASER : Bool := FALSE;   // A FAULT MESSAGE OF THE LASER DEVICE IS ACTIVE
            MONITORING : Bool := FALSE;   // A MONITORING MESSAGE OF THE LASER DEVICE IS ACTIVE
            SIK_OPEN : Bool := FALSE;   // THE SAFETY CIRCUIT (SIK) IS OPEN
            SET_3 : Bool := FALSE;   // SET OUTPUTS 3
            SET_2 : Bool := FALSE;   // SET OUTPUTS 2
            SET_1 : Bool := FALSE;   // SET OUTPUTS 1
            PROG_CANCELED : Bool := FALSE;   // LASER PROGRAM HAS BEEN CANCELLED
            PROG_COMPLETED : Bool := FALSE;   // LASER PROGRAM IS COMPLETED
            PROG_ACTIVE : Bool := FALSE;   // LASER PROGRAM IS ACTIVE
            LASER_READY : Bool := FALSE;   // THE LASER OF THE LASER DEVICE IS READY
            LASER_IS_ON : Bool := FALSE;   // THE LASER OF THE LASER DEVICE IS SWITCHED ON
            EXT_ACTIV_ACTIVE : Bool := FALSE;   // EXTERNAL ACTIVATION IS ACTIVE
         END_STRUCT;
         PROGRAMNO_ACK : Byte := B#16#0;   // ACKNOWLEDGEMENT OF THE NUMBER OF THE LASER PROGRAMSELECTED
         LIGHTPATH_ACK : Byte := B#16#0;   // ACKNOWLEDGEMENT OF THE NUMBER OF THE CURRENTLY SET LIGHTPATH
         SHUTTER_SWITCH_1 : Bool;   // POSITION OF THE SHUTTER SWITCHES
         SHUTTER_SWITCH_2 : Bool;   // POSITION OF THE SHUTTER SWITCHES
         SHUTTER_SWITCH_3 : Bool;   // POSITION OF THE SHUTTER SWITCHES
         SHUTTER_SWITCH_4 : Bool;   // POSITION OF THE SHUTTER SWITCHES
         SHUTTER_SWITCH_5 : Bool;   // POSITION OF THE SHUTTER SWITCHES
         SHUTTER_SWITCH_6 : Bool;   // POSITION OF THE SHUTTER SWITCHES
         SHUTTER_SWITCH_7 : Bool;   // POSITION OF THE SHUTTER SWITCHES
         SHUTTER_SWITCH_8 : Bool;   // POSITION OF THE SHUTTER SWITCHES
         FAULT_SLOT : Bool := FALSE;   // A LOCAL FAULT HAS OCCURRED FOR THIS SLOT
         MONITORING_SLOT : Bool := FALSE;   // A LOCAL MONITORING HAS OCCURRED FOR THIS SLOT
         RESERVED_1 : Bool := FALSE;   // RESERVE
         OPTICS_AVAILABLE : Bool := FALSE;   // FOCUSING OPTICS OR LIGHT PATH COMPONENT IS ENABLED.
         OPTICS_READY : Word;   // THE FOCUSING OPTICS OR LIGHT PATH COMPONENT IS READY FOR OPERATION.
         VALUES_IN_RANGE : Bool := FALSE;   // APPLICATION VALUES CROSSJET PRESSURE, EXHAUSTION AND SHIELDING GAS ARE IN THE ADMISSIBLE RANGE
         PROT_GLASS_CONTAM : Bool := FALSE;   // LIMIT VALUE MAX1 OF THE PROTECTIVE GLASS CONTAMINATION HASBEEN REACHED
         PROT_GLASS_LIFE_RCHD : Bool := FALSE;   // LIMIT VALUE MAX2 OF THE PROTECTIVE GLASS CONTAMINATION HASBEEN REACHED
         MEAS_VAL_OUT_ACT : Bool := FALSE;   // OUTPUT WORD 4 OUTPUTS MEASURED VALUE ID
         MAINTENACE : Bool := FALSE;   // MAINTENANCE OF THE LASER DEVICE IS REQUIRED
         RESERVED_2 : Bool;   // RESERVE
         CALIBRATION : Bool := FALSE;   // THE LASER IS BEING CALIBRATED OR LASER SELFTEST IS ACTIVE
         ALIVE_TICK : Bool := FALSE;   // LASER CONTROL IS ACTIVE
         EXT_COOL_ON : Bool := FALSE;   // EXTERNAL COOLING CIRCUIT IS SWITCHED ON OR THE LASER DEVICE REQUIRES COOLING WATER
         RESERVED_3 : Bool;   // RESERVE
         RESERVED_4 : Bool;   // RESERVE
         LASER_NO_1 : Bool;   // NUMBER OF THE LASER DEVICE BIT 1
         LASER_NO_2 : Bool;   // NUMBER OF THE LASER DEVICE BIT 2
         LASER_NO_3 : Bool;   // NUMBER OF THE LASER DEVICE BIT 3
         LASER_NO_4 : Bool;   // NUMBER OF THE LASER DEVICE BIT 4
         LASER_NO_5 : Bool;   // NUMBER OF THE LASER DEVICE BIT 5
         LASER_NO_6 : Bool;   // NUMBER OF THE LASER DEVICE BIT 6
         LASER_NO_7 : Bool;   // NUMBER OF THE LASER DEVICE BIT 7
         LASER_NO_8 : Bool;   // NUMBER OF THE LASER DEVICE BIT 8
         MESSAGE_NUM : Byte;   // MESSAGE CODE NUM
         MESSAGE_ID : Byte;   // MESSAGE CODE ID
         MESSAGE_CODE : Word;   // MESSAGE CODE OF THE REPORTING COMPONENT
         LASER_POWER : Word;   // CW LASER: LASER POWER
         ENERGY : Word;   // PULSE ENERGY
         RESERVED_WORD_8 : Word;   // RESERVE WORD
      END_STRUCT;
   END_STRUCT;
END_TYPE

TYPE "LASER ACTIVE"
// stored: IsFailsafeCompliant false
   STRUCT
      "EMISSION LASER STILL PERMANENT CONDITIONS" : Bool;
      "EMISSION LASER STILL ENABLE REQUEST" : Bool;
      "EMISSION LASER STILL DISABLE REQUEST" : Bool;
      "EMISSION LASER STILL ENABLE MODE" : Bool;
      "LASER ACTIVE A" : Bool;
      "LASER ACTIVE START GENERAL CONDITIONS" : Bool;
      "LASER ACTIVE START INITIAL CONDITIONS" : Bool;
      "LASER ACTIVE MANUAL START REQUEST" : Bool;
      "LASER ACTIVE AUTO START REQUEST" : Bool;
      "LASER ACTIVE START REQUEST" : Bool;
      "LASER ACTIVE START COMMAND" : Bool;
      "LASER ACTIVE LASER ACTIVE ON" : Bool;
      "LASER ACTIVE FEEDBACK ON" : Bool;
      "LASER ACTIVE STOP GENERAL CONDITIONS" : Bool;
      "LASER ACTIVE STOP INITIAL CONDITIONS" : Bool;
      "LASER ACTIVE MANUAL STOP REQUEST" : Bool;
      "LASER ACTIVE AUTO STOP REQUEST" : Bool;
      "LASER ACTIVE STOP REQUEST" : Bool;
      "LASER ACTIVE STOP COMMAND" : Bool;
      "LASER ACTIVE STOPPED" : Bool;
      "LASER ACTIVE FEEDBACK OFF" : Bool;
      "LASER ACTIVE PROGRAM NOT ACTIVE" : Bool;
      "LASER ACTIVE WARNING GONE" : Bool;
      "LASER ACTIVE START GENERAL CONDITION HELP" : Bool;
      "LASER ACTIVE START INITIAL CONDITION HELP" : Bool;
      "LASER ACTIVE STOP GENERAL CONDITION HELP" : Bool;
      "LASER ACTIVE STOP INITIAL CONDITION HELP" : Bool;
      "LASER ACTIVE FAULT" : Bool;
   END_STRUCT;
END_TYPE

TYPE "LASER POINTER"
// stored: IsFailsafeCompliant false
   STRUCT
      "LASER POINTER INPUT ON" : Bool;
      "LASER POINTER START GENERAL CONDITIONS" : Bool;
      "LASER POINTER START INITIAL CONDITIONS" : Bool;
      "LASER POINTER MANUAL START REQUEST" : Bool;
      "LASER POINTER AUTO START REQUEST" : Bool;
      "LASER POINTER START REQUEST" : Bool;
      "LASER POINTER START COMMAND" : Bool;
      "LASER POINTER LASER SYSTEM ON" : Bool;
      "LASER POINTER FEEDBACK ON" : Bool;
      "LASER POINTER STOP GENERAL CONDITIONS" : Bool;
      "LASER POINTER STOP INITIAL CONDITIONS" : Bool;
      "LASER POINTER MANUAL STOP REQUEST" : Bool;
      "LASER POINTER AUTO STOP REQUEST" : Bool;
      "LASER POINTER STOP REQUEST" : Bool;
      "LASER POINTER STOP COMMAND" : Bool;
      "LASER POINTER STOPPED" : Bool;
      "LASER POINTER FEEDBACK OFF" : Bool;
      "LASER POINTER WARNING GONE" : Bool;
      "LASER POINTER START GENERAL CONDITION HELP" : Bool;
      "LASER POINTER START INITIAL CONDITION HELP" : Bool;
      "LASER POINTER STOP GENERAL CONDITION HELP" : Bool;
      "LASER POINTER STOP INITIAL CONDITION HELP" : Bool;
      "LASER POINTER NOT READY ALARM" : Bool;
      "LASER POINTER FAULT" : Bool;
   END_STRUCT;
END_TYPE

TYPE "LASER READY"
// stored: IsFailsafeCompliant false
   STRUCT
      "LASER READY LASER ARM INPUT ACKNOWLEDGE_1" : Bool;
      "LASER READY INPUT LASER EMERGENCY STOP" : Bool;
      "LASER READY INPUT LASER SC STATUS" : Bool;
      "LASER READY CIRCUIT BREAKER" : Bool;
      "LASER READY" : Bool;
      "LASER READY START GENERAL CONDITIONS" : Bool;
      "LASER READY START INITIAL CONDITIONS" : Bool;
      "LASER READY MANUAL START REQUEST" : Bool;
      "LASER READY AUTO START REQUEST" : Bool;
      "LASER READY START REQUEST" : Bool;
      "LASER READY START COMMAND" : Bool;
      "LASER READY LASER SYSTEM ON" : Bool;
      "LASER READY FEEDBACK ON" : Bool;
      "LASSER ANALOG CONTROL ACTIVE" : Bool;
      "LASER READY STOP GENERAL CONDITIONS" : Bool;
      "LASER READY STOP INITIAL CONDITIONS" : Bool;
      "LASER READY MANUAL STOP REQUEST" : Bool;
      "LASER READY AUTO STOP REQUEST" : Bool;
      "LASER READY STOP REQUEST" : Bool;
      "LASER READY STOP COMMAND" : Bool;
      "LASER READY STOPPED" : Bool;
      "LASER READY FEEDBACK OFF" : Bool;
      "LASER READY CIRCUIT BREAKER ALARM" : Bool;
      "LASER READY LASER ERROR" : Bool;
      "LASER READY WARNING LASER" : Bool;
      "LASER READY LASER NOT READY" : Bool;
      "LASER READY LASER NOT SWITCHED ON" : Bool;
      "LASER READY FAULT" : Bool;
      "LASER READY WARNING GONE" : Bool;
      "LASER READY START GENERAL CONDITION HELP" : Bool;
      "LASER READY START INITIAL CONDITION HELP" : Bool;
      "LASER READY STOP GENERAL CONDITION HELP" : Bool;
      "LASER READY STOP INITIAL CONDITION HELP" : Bool;
      "LASER MIN POWER LIMIT" : Int;
      "LASER MAX POWER LIMIT" : Int;
      "LASER POWER COMMAND" : Int;
      "TIMER AUTO REQ ON" : TON_TIME;
      "TIMER FAULT 1" { S7_SetPoint := 'True'} : TON_TIME;
      "TIMER FAULT 2" { S7_SetPoint := 'True'} : TON_TIME;
      "TIMER FAULT 3" { S7_SetPoint := 'True'} : TON_TIME;
      "TIMER LASER REQUEST" { S7_SetPoint := 'True'} : TON_TIME;
      "TIMER REST ERROR" { S7_SetPoint := 'True'} : TON_TIME;
   END_STRUCT;
END_TYPE

TYPE "COOLING_SENSOR"
// stored: IsFailsafeCompliant false
   STRUCT
      COOLING_FLOW_SENSOR_ACTUAL_VALUE : Real;   // COOLING FLOW SENSOR VALUE
      COOLING_TEMP_SENSOR_ACTUAL_VALUE : Real;   // COOLING TEMPERATURE SENSOR VALUE
      COOLING_FLOW_LOW_WARNING_HMI_VALUE : Real := 3.2;   // COOLING FLOW LOW WARNING VALUE
      COOLING_FLOW_HIGH_WARNING_HMI_VALUE : Real := 4.8;   // COOLING FLOW HIGH WARNING VALUE
      COOLING_FLOW_LOW_ALARM_HMI_VALUE : Real := 3.2;   // COOLING FLOW LOW ALARM VALUE
      COOLING_FLOW_HIGH_ALARM_HMI_VALUE : Real := 6.0;   // COOLING FLOW HIGH ALARM VALUE
      COOLING_TEMP_LOW_WARNING_HMI_VALUE : Real := 27.0;   // COOLING TEMPERATURE LOW WARNING VALUE
      COOLING_TEMP_HIGH_WARNING_HMI_VALUE : Real := 40.0;   // COOLING TEMPERATURE HIGH WARNING VALUE
      COOLING_TEMP_LOW_ALARM_HMI_VALUE : Real := 27.0;   // COOLING TEMPERATURE LOW ALARM VALUE
      COOLING_TEMP_HIGH_ALARM_HMI_VALUE : Real := 40.0;   // COOLING TEMPERATURE HIGH ALARM VALUE
   END_STRUCT;
END_TYPE

TYPE "LASER GUIDE"
// stored: IsFailsafeCompliant false
   STRUCT
      START_GENERAL_CONDITIONS : Bool;   // Start General Conditions
      START_GENERAL_CONDITIONS_HELP : Bool;   // Start General Conditions Help
      START_INITIAL_CONDITIONS : Bool;   // Start Initial Conditions
      START_INITIAL_CONDITIONS_HELP : Bool;   // Start Initial Conditions Help
      START_MANUAL_REQUEST : Bool;   // Start Manual Request
      FEEDBACK_ON : Bool;   // Feedback On
      START_AUTO_REQUEST : Bool;   // Start Auto Request
      START_GLOBAL_REQUEST : Bool;   // Start Global Request
      START_COMMAND : Bool;   // Start Command
      LASER_ON : Bool;   // Laser On
      STOP_GENERAL_CONDITIONS : Bool;   // Stop General Conditions
      STOP_GENERAL_CONDITIONS_HELP : Bool;   // Stop General Conditions Help
      STOP_INITIAL_CONDITIONS : Bool;   // Stop Initial Conditions
      STOP_INITIAL_CONDITIONS_HELP : Bool;   // Stop Initial Conditions Help
      STOP_MANUAL_REQUEST : Bool;   // Manual Stop Request
      STOP_AUTO_REQUEST : Bool;   // Auto Stop Request
      STOP_GLOBAL_REQUEST : Bool;   // Stop Global Request
      STOP_COMMAND : Bool;   // Stop Command
      STOPPED : Bool;   // Stopped
      FEEDBACK_OFF : Bool;   // Feedback Off
      LASER_FAULT : Bool;   // Laser Faulted
   END_STRUCT;
END_TYPE

TYPE "PYROCONTROL"
// stored: IsFailsafeCompliant false
   STRUCT
      INPUT_PYROMETER : Real;   // Input Pyrometer
      PYROMETER_ACTUAL_TEMP : Real;   // Pyrometer Actual Temp
      MAX_POWER : Real;   // HMI Max Power
      UNMODIFIED_POWER : Real;   // Unmodified Power
      POWER_RATIO : Real;   // Power Ratio
      MODIFIED_POWER : Real;   // Modified Power
      COMMANDED_POWER : Int;   // Commanded Power
      REAL_POWER : Int;   // Real Power
   END_STRUCT;
END_TYPE

TYPE "PYROMETER"
// stored: IsFailsafeCompliant false
   STRUCT
      PYROMETER_READY_INPUT : Bool;   // Pyrometer Ready Input
      PYROMETER_FAULT_INPUT : Bool;   // Pyrometer Fault Input
      START_GENERAL_CONDITIONS : Bool;   // Start General Conditions
      START_INITIAL_CONDITIONS : Bool;   // Start Initial Conditions
      START_MANUAL_REQUEST : Bool;   // Start Manual Request
      START_AUTO_REQUEST : Bool;   // Start Auto Request
      START_GLOBAL_REQUEST : Bool;   // Start Global Request
      START_COMMAND : Bool;   // Start Command
      STARTED : Bool;   // Started
      FEEDBACK_STARTED : Bool;   // Feedback Started
      STOP_GENERAL_CONDITIONS : Bool;   // Stop General Conditions
      STOP_INITIAL_CONDITIONS : Bool;   // Stop Initial Conditions
      STOP_MANUAL_REQUEST : Bool;   // Stop Manual Request
      STOP_AUTO_REQUEST : Bool;   // Stop Auto Request
      STOP_GLOBAL_REQUEST : Bool;   // Stop Global Request
      STOP_COMMAND : Bool;   // Stop Command
      STOPPED : Bool;   // Stopped
      FEEDBACK_STOP : Bool;   // Feedback Stop
      SPARE_BYTE_4 : Byte;   // Spare Byte 4
      DIFERENCIAL_PROTECTION_FAULT : Bool;   // Diferential Protection Fault
      CIRCUIT_BRAKER_FAULT : Bool;   // Circuit Breaker Fault
      CONTACTOR_FEEDBACK_FAULT : Bool;   // Contactor Feedback Fault
      SAFETY_FEEDBACK_FAULT : Bool;   // Safety Feedback Fault
      FEEDBACK_FAULT : Bool;   // Feedback Fault
      ERROR_FAULT : Bool;   // Error Fault
      NOT_RUNNING_ALARM : Bool;   // Not Running Alarm
      PRESSURE_1 : Bool;   // Pressure_1
      AUX0 : Bool;   // Aux0
      AUX1 : Bool;   // Aux1
      AUX2 : Bool;   // Aux2
      AUX3 : Bool;   // Aux3
      WARNING_GONE : Bool;   // Warning Gone
      AUX5 : Bool;   // Aux5
      AUX6 : Bool;   // Aux6
      AUX7 : Bool;   // Aux7
      START_GENERAL_CONDITIONS_HELP : Bool;   // Start General Conditions Help
      START_INITIAL_CONDITIONS_HELP : Bool;   // Start Initial Conditions Help
      STOP_GENERAL_CONDITIONS_HELP : Bool;   // Stop General Conditions Help
      STOP_INITIAL_CONDITIONS_HELP : Bool;   // Stop Initial Conditions Help
      FAULT : Bool;   // Fault
   END_STRUCT;
END_TYPE

DATA_BLOCK "DB2001_MODES_FEEDERS"   // DB2001
{ S7_Optimized_Access := 'FALSE'; DB_Accessible_From_OPC_UA := 'FALSE' }
AUTHOR : ETXETAR
VERSION : 1.0
// stored: AutoNumber false, DBAccessibleFromOPCUA false, DBAccessibleFromWebserver true, IsOnlyStoredInLoadMemory false, IsWriteProtectedInAS false
   VAR RETAIN
      GENERAL : "AUTO_SINGLE_SEMI_MANUAL";
   END_VAR
BEGIN
END_DATA_BLOCK

DATA_BLOCK "DB2002_MODES_HOPPERS"   // DB2002
{ S7_Optimized_Access := 'FALSE'; DB_Accessible_From_OPC_UA := 'FALSE' }
AUTHOR : ETXETAR
VERSION : 1.0
// stored: AutoNumber false, DBAccessibleFromOPCUA false, DBAccessibleFromWebserver true, IsOnlyStoredInLoadMemory false, IsWriteProtectedInAS false
   VAR RETAIN
      GENERAL : "AUTO_SINGLE_SEMI_MANUAL";
   END_VAR
BEGIN
END_DATA_BLOCK

DATA_BLOCK "DB2031_CYCLES_GENERAL"   // DB2031
{ S7_Optimized_Access := 'FALSE'; DB_Accessible_From_OPC_UA := 'FALSE' }
AUTHOR : ETXETAR
VERSION : 1.0
// stored: AutoNumber false, DBAccessibleFromOPCUA false, DBAccessibleFromWebserver true, IsOnlyStoredInLoadMemory false, IsWriteProtectedInAS false
   VAR RETAIN
      DRY_CYCLE { S7_SetPoint := 'True'} : "CYCLES";
      MANUAL_LOAD_CYCLE { S7_SetPoint := 'True'} : "CYCLES";
   END_VAR
BEGIN
   // DRY_CYCLE.CYCLE_SELECTED : DRY CYCLE SELECTED
   // DRY_CYCLE.CYCLE_COMPLETED : DRY CYCLE COMPLETED
   // MANUAL_LOAD_CYCLE.CYCLE_SELECTED : MANUAL LOAD CYCLE SELECTED
   // MANUAL_LOAD_CYCLE.CYCLE_COMPLETED : MANUAL LOAD CYCLE COMPLETED
END_DATA_BLOCK

DATA_BLOCK "DB2100_GENERAL"   // DB2100
{ S7_Optimized_Access := 'FALSE'; DB_Accessible_From_OPC_UA := 'FALSE' }
AUTHOR : ETXETAR
VERSION : 1.0
// stored: AutoNumber false, DBAccessibleFromOPCUA false, DBAccessibleFromWebserver true, IsOnlyStoredInLoadMemory false, IsWriteProtectedInAS false
   VAR RETAIN
      EMERGENCY_STOP_ACTIVE : Bool;   // EMERGENCY STOP PILZ / EMERGENCY STOP ACTIVE
      SAFETY_GATES_CLOSED_LOCKED : Bool;   // GATES CLOSED & LOCKED PILZ / SAFETY GATES CLOSED AND LOCKED
      MACHINE_READY_POWER_ENABLED : Bool;   // MACHINE READY PILZ / MACHINE READY POWER ENABLED
      ANY_AXIS_OR_CH_BYPASSED : Bool;   // ANY AXIS BYPASSED / ANY AXIS OR CHANNEL BYPASSED
      ANY_AXIS_OR_CH_BYPASSED_ALARM : Bool;   // ANY AXIS BYPASSED FAULT / ANY AXIS OR CHANNEL BYPASSED ALARM
      PROGRAMMING_ALARM : Bool;   // ANY PROGRAMMING ALARM
      BYPASS_SAFETY_DOORS_ENABLED : Bool;   // BYPASS SAFETY DOORS ENABLE / BYPASS SAFETY DOORS ENABLED
      BA1_OR_BA3_MODE_ENABLED : Bool;   // BA1 OR BA3 MODE ENABLED
      ANY_BA_MODE_ENABLED : Bool;   // ANY BA MODE ENABLED
      CHECKSUM_OK : Bool;   // CITI Checksum Overall OK / CHECKSUM OK
      EMERGENCY_STOP_ACTIVE_ALARM : Bool;   // EMERGENCY STOP ACTIVE / EMERGENCY STOP ACTIVE ALARM
      OVERRIDE_LOWER_THAN_80 : Bool;   // OVERRIDE LOWER THAN 80
      OVERRIDE_100 : Bool;   // OVERRIDE 100
      WARNINGS_GONE : Bool;   // UTILITY SKIDS WARNINGS GONE
      CHECK_NETWORK_LOGIC_ALARM : Bool;   // CHECK NETWORK LOGIC ALARM
   END_VAR
BEGIN
END_DATA_BLOCK

DATA_BLOCK "DB2130_TIMERS"   // DB2130
{ S7_Optimized_Access := 'FALSE'; DB_Accessible_From_OPC_UA := 'FALSE' }
AUTHOR : ETXETAR
VERSION : 1.0
// stored: AutoNumber false, DBAccessibleFromOPCUA false, DBAccessibleFromWebserver true, IsOnlyStoredInLoadMemory false, IsWriteProtectedInAS false
   VAR
      TIMER_CH2_ACK_M50 { S7_SetPoint := 'True'} : IEC_TIMER;   // CHANNEL 2 ACKNOWLEDGE M50 TIMER
      TIMER_CH2_ACK_M51 { S7_SetPoint := 'True'} : IEC_TIMER;   // CHANNEL 2 ACKNOWLEDGE M51 TIMER
      TIMER_CH2_ACK_M160 { S7_SetPoint := 'True'} : IEC_TIMER;   // CHANNEL 2 ACKNOWLEDGE M160 TIMER
      TIMER_CH3_ACK_M50 { S7_SetPoint := 'True'} : IEC_TIMER;   // CHANNEL 3 ACKNOWLEDGE M50 TIMER
      TIMER_CH3_ACK_M51 { S7_SetPoint := 'True'} : IEC_TIMER;   // CHANNEL 3 ACKNOWLEDGE M51 TIMER
      TIMER_CH3_ACK_M160 { S7_SetPoint := 'True'} : IEC_TIMER;   // CHANNEL 3 ACKNOWLEDGE M160 TIMER
   END_VAR
BEGIN
   TIMER_CH2_ACK_M50.PT := T#2s;
   TIMER_CH2_ACK_M51.PT := T#2s;
   TIMER_CH2_ACK_M160.PT := T#1s;
   TIMER_CH3_ACK_M50.PT := T#2s;
   TIMER_CH3_ACK_M51.PT := T#2s;
   TIMER_CH3_ACK_M160.PT := T#1s;
END_DATA_BLOCK

DATA_BLOCK "DB2101_LINE_CONTACTOR"   // DB2101
{ S7_Optimized_Access := 'FALSE'; DB_Accessible_From_OPC_UA := 'FALSE' }
AUTHOR : ETXETAR
VERSION : 1.0
// stored: AutoNumber false, DBAccessibleFromOPCUA false, DBAccessibleFromWebserver true, IsOnlyStoredInLoadMemory false, IsWriteProtectedInAS false
   VAR
      FEEDBACK_IN_1 : Bool;   // CONTACTOR FEEDBACK INPUT 1
      FEEDBACK_IN_2 : Bool;   // CONTACTOR FEEDBACK INPUT 2
      LINE_CONTACTOR_ENABLED : Bool;   // LINE CONTACTOR ENABLED
      ON_GENERAL_CONDITIONS : Bool;   // UNIT 01L CYCLE SEQUENCE GENERAL CONDITIONS / SWITCH ON GENERAL CONDITIONS
      ON_INITIAL_CONDITIONS : Bool;   // UNIT 01L CYCLE SEQUENCE INITIAL CONDITIONS / SWITCH ON INITIAL CONDITIONS
      ON_REQ_1 : Bool;   // UNIT 01L CYCLE SEQUENCE STEP 4 / SWITCH ON REQUEST 1
      ON_REQ_2 : Bool;   // UNIT 01L CYCLE SEQUENCE STEP 5 / SWITCH ON REQUEST 2
      ON_REQ_3 : Bool;   // UNIT 01L CYCLE SEQUENCE STEP 6 / SWITCH ON REQUEST 3
      ON_REQ_4 : Bool;   // UNIT 01L CYCLE SEQUENCE STEP 7 / SWITCH ON REQUEST 4
      OFF_GENERAL_CONDITIONS : Bool;   // UNIT 01L CYCLE SEQUENCE GENERAL CONDITIONS / SWITCH OFF GENERAL CONDITIONS
      OFF_INITIAL_CONDITIONS : Bool;   // UNIT 01L CYCLE SEQUENCE INITIAL CONDITIONS / SWITCH OFF INITIAL CONDITIONS
      OFF_REQ_1 : Bool;   // UNIT 01L CYCLE SEQUENCE STEP 4 / SWITCH OFF REQUEST 1
      OFF_REQ_2 : Bool;   // UNIT 01L CYCLE SEQUENCE STEP 5 / SWITCH OFF REQUEST 2
      OFF_REQ_3 : Bool;   // UNIT 01L CYCLE SEQUENCE STEP 6 / SWITCH OFF REQUEST 3
      OFF_REQ_4 : Bool;   // UNIT 01L CYCLE SEQUENCE STEP 7 / SWITCH OFF REQUEST 4
      STEP_1_CONTACTOR_ON : Bool;   // UNIT 01L CYCLE SEQUENCE STEP 1 / STEP 1
      STEP_2_POWER_SUPPLY_ON : Bool;   // UNIT 01L CYCLE SEQUENCE STEP 2 / STEP 2
      STEP_3_OFF3_ON : Bool;   // UNIT 01L CYCLE SEQUENCE STEP 3 / STEP 3
      STEP_4 : Bool;   // UNIT 01L CYCLE SEQUENCE STEP 8 / STEP 4
      STEP_5 : Bool;   // UNIT 01L CYCLE SEQUENCE STEP 9 / STEP 5
      STEP_6 : Bool;   // UNIT 01L CYCLE SEQUENCE STEP 10 / STEP 6
      STEP_7 : Bool;   // UNIT 01L CYCLE SEQUENCE STEP 11 / STEP 7
      FEEDBACK_1_ALM : Bool;   // CONTACTOR FEEDBACK 1 ALARM
      FEEDBACK_2_ALM : Bool;   // CONTACTOR FEEDBACK 2 ALARM
      O_LINE_CONTACTOR_1 : Bool;   // UNIT 01L CYCLE SEQUENCE AUX0 / OPTION LINE CONTACTOR 1
      O_LINE_CONTACTOR_2 : Bool;   // UNIT 01L CYCLE SEQUENCE AUX1 / OPTION LINE CONTACTOR 2
      AUX2 : Bool;   // UNIT 01L CYCLE SEQUENCE AUX2 / AUXILIARY 2
      AUX3 : Bool;   // UNIT 01L CYCLE SEQUENCE AUX3 / AUXILIARY 3
      AUX5 : Bool;   // UNIT 01L CYCLE SEQUENCE AUX5 / AUXILIARY 5
      AUX6 : Bool;   // UNIT 01L CYCLE SEQUENCE AUX6 / AUXILIARY 6
      AUX7 : Bool;   // UNIT 01L CYCLE SEQUENCE AUX7 / AUXILIARY 7
      AUX8 : Bool;   // UNIT 01L CYCLE SEQUENCE AUX7 / AUXILIARY 8
      NOT_SWITCHED_ON_WARNING : Bool;   // LINE CONTACTOR NOT SWITCHED ON WARNING
      GENERAL_CONDITIONS_HELP : Bool;   // UNIT 01L CYCLE SEQUENCE GENERAL CONDITIONS HELP / GENERAL CONDITIONS HELP
      INITIAL_CONDITIONS_HELP : Bool;   // UNIT 01L CYCLE SEQUENCE INITIAL CONDITIONS HELP / INITIAL CONDITIONS HELP
      ANY_ACTIVE_ALARM : Bool;   // ANY ACTIVE ALARM
      IS_ALARMS : Bool;   // IMMEDIATE STOP ALARMS
      WARNINGS : Bool;   // WARNINGS
      WARNINGS_GONE : Bool;   // UNIT 01L CYCLE SEQUENCE PREALARM GONE / WARNINGS GONE
      TIMER_CONTACTOR_LINE_FEEDBACK_1 : TON_TIME;   // CONTACTOR LINE FEEDBACK 1 TIMER
      TIMER_CONTACTOR_LINE_FEEDBACK_2 : TON_TIME;   // CONTACTOR LINE FEEDBACK 2 TIMER
      TIMER_STEP_2_START_ON : TON_TIME;   // STEP 1 START ON TIMER
      TIMER_STEP_3_START_ON : TON_TIME;   // STEP 2 START ON TIMER
      TIMER_EMERGENCY_STOP_PILZ_REQUEST : TON_TIME;   // EMERGENCY STOP PILZ REQUEST TIMER
      TIMER_START_OFF_REQUEST_2 : TOF_TIME;   // START OFF REQUEST 1 TIMER
      TIMER_START_OFF_REQUEST_3 : TOF_TIME;   // START OFF REQUEST 2 TIMER
   END_VAR
BEGIN
   TIMER_CONTACTOR_LINE_FEEDBACK_1.PT := T#500ms;
   TIMER_CONTACTOR_LINE_FEEDBACK_2.PT := T#500ms;
   TIMER_STEP_2_START_ON.PT := T#1s;
   TIMER_STEP_3_START_ON.PT := T#100ms;
   TIMER_EMERGENCY_STOP_PILZ_REQUEST.PT := T#5s;
   TIMER_START_OFF_REQUEST_2.PT := T#1s;
   TIMER_START_OFF_REQUEST_3.PT := T#1s;
END_DATA_BLOCK

DATA_BLOCK "DB2102_INFEED_MODULE"   // DB2102
{ S7_Optimized_Access := 'FALSE'; DB_Accessible_From_OPC_UA := 'FALSE' }
AUTHOR : ETXETAR
VERSION : 1.0
// stored: AutoNumber false, DBAccessibleFromOPCUA false, DBAccessibleFromWebserver true, IsOnlyStoredInLoadMemory false, IsWriteProtectedInAS false
   VAR RETAIN
      INFEED_MODULE_1_READY_I : Bool;   // INPUT 611D READY / INFEED MODULE 1 READY INPUT
      INFEED_MODULE_1_ENABLED_I : Bool;   // INPUT 611D ENABLED / INFEED MODULE 1 ENABLED INPUT
      INFEED_MODULE_1_OVERTEMPERATURE_I : Bool;   // INPUT 611D OVERTEMPERATURE / INFEED MODULE 1 OVERTEMPERATURE INPUT
      INFEED_MODULE_2_READY_I : Bool;   // INPUT 611D READY / INFEED MODULE 2 READY INPUT
      INFEED_MODULE_2_ENABLED_I : Bool;   // INPUT 611D ENABLED / INFEED MODULE 2 ENABLED INPUT
      INFEED_MODULE_2_OVERTEMPERATURE_I : Bool;   // INPUT 611D OVERTEMPERATURE / INFEED MODULE 2 OVERTEMPERATURE INPUT
      INFEED_MODULE_READY : Bool;   // POWER SUPPLY 611D READY / INFEED MODULE READY
      INFEED_MODULE_READY_ENABLE_AXES : Bool;   // POWER SUPPLY READY ENABLE AXIS / INFEED MODULE READY ENABLE AXIS
      INFEED_MODULE_1_NOT_READY_ALARM : Bool;   // POWER SUPPLY 611D NOT READY / INFEED MODULE 1 NOT READY ALARM
      INFEED_MODULE_1_OVERTEMPERATURE_ALARM : Bool;   // POWER SUPPLY 611D OVERTEMPERATURE / INFEED MODULE 1 OVERTEMPERATURE ALARM
      INFEED_MODULE_2_NOT_READY_ALARM : Bool;   // POWER SUPPLY 611D NOT READY / INFEED MODULE 2 NOT READY ALARM
      INFEED_MODULE_2_OVERTEMPERATURE_ALARM : Bool;   // POWER SUPPLY 611D OVERTEMPERATURE / INFEED MODULE 2 OVERTEMPERATURE ALARM
      NCU_HEAT_SINK_TEMPERATURE_ALARM : Bool;   // NCU TEMPERATURE FAULT / NCU HEAT SINK TEMPERATURE ALARM
      NCU_LOW_BATTERY_ALARM : Bool;   // NC BATTERY LOW / NCU LOW BATTERY ALARM
      NCU_AIR_TEMPERATURE_ALARM : Bool;   // HEAT SINK AIR FLOW FAULT / NCU AIR TEMPERATURE ALARM
      NCK_ALARM : Bool;   // NCK ALARM
      ANY_ACTIVE_ALARM : Bool;   // ANY ACTIVE ALARM
      IS_ALARMS : Bool;   // IMMEDIATE STOP ALARMS
      SEOC_ALARMS : Bool;   // STOP AT END OF CYCLE ALARMS
      INFEED_MODULE_1_NOT_READY_AUX : Bool;   // AUXILIARY NOT READY / INFEED MODULE 1 NOT READY AUXILIARY
      INFEED_MODULE_2_NOT_READY_AUX : Bool;   // AUXILIARY NOT READY / INFEED MODULE 2 NOT READY AUXILIARY
      TIMER_INFEED_MODULE_READY : TOF_TIME;   // INFEED MODULE READY TIMER
      TIMER_INFEED_MODULE_1_NOT_READY : TON_TIME;   // INFEED MODULE 1 NOT READY TIMER
      TIMER_INFEED_MODULE_2_NOT_READY : TON_TIME;   // INFEED MODULE 2 NOT READY TIMER
      TIMER_NCK_ALAR_DELAY { S7_SetPoint := 'True'} : TON_TIME;   // NCK ALARM TIMER
   END_VAR
BEGIN
   TIMER_INFEED_MODULE_READY.PT := T#1s;
   TIMER_INFEED_MODULE_1_NOT_READY.PT := T#200ms;
   TIMER_INFEED_MODULE_2_NOT_READY.PT := T#200ms;
   TIMER_NCK_ALAR_DELAY.PT := T#100ms;
END_DATA_BLOCK

DATA_BLOCK "DB2103_ELECTRICAL_CABINET"   // DB2103
{ S7_Optimized_Access := 'FALSE'; DB_Accessible_From_OPC_UA := 'FALSE' }
AUTHOR : ETXETAR
VERSION : 1.0
// stored: AutoNumber false, DBAccessibleFromOPCUA false, DBAccessibleFromWebserver true, IsOnlyStoredInLoadMemory false, IsWriteProtectedInAS false
   VAR RETAIN
      INPUT_230_VAC_BREAKER : Bool;   // MAIN CABINET CIRCUIT BREAKER TRIPPED / INPUT 230 VAC CABINET CIRCUIT BREAKER TRIPPED
      INPUT_AIR_UNIT_1_BREAKER : Bool;   // AIR UNIT BREAKER - STOP END OF CYCLE / INPUT AIR UNIT 1 CRICUIT BREAKER TRIPPED
      INPUT_AIR_UNIT_2_BREAKER : Bool;   // AIR UNIT BREAKER - STOP END OF CYCLE / INPUT AIR UNIT 2 CIRCUIT BREAKER TRIPPED
      INPUT_24VDC_BREAKER_1 : Bool;   // CIRCUIT BREAKER 24 V DC / INPUT 24 VDC CIRCUIT BREAKER TRIPPED 1
      INPUT_24VDC_BREAKER_2 : Bool;   // CIRCUIT BREAKER 24 V DC / INPUT 24 VDC CIRCUIT BREAKER TRIPPED 2
      INPUT_FC35_1_BREAKER : Bool;   // INPUT BREAKER 3004 / INPUT FC35.1 CIRCUIT BREAKER TRIPPED
      INPUT_FC35_2_BREAKER : Bool;   // INPUT FC35.2 CIRCUIT BREAKER TRIPPED
      INPUT_FC35_3_BREAKER : Bool;   // INPUT FC35.3 CIRCUIT BREAKER TRIPPED
      INPUT_SINAMICS_BREAKER : Bool;   // SINAMICS CIRCUIT BREAKER TRIPPED INPUT / INPUT SINAMICS CIRCUIT BREAKER TRIPPED
      "INPUT_110/120/220/230VAC_BREAKER" : Bool;   // CIRCUIT BREAKER F1 - F4 / INPUT 110/120/220/230VAC CIRCUIT BREAKER TRIPPED
      INPUT_SINAMICS_BREAKER_1 : Bool;   // INPUT SINAMICS CIRCUIT BREAKER TRIPPED
      INPUT_CAB_LIGHT_BREAKER : Bool;   // CIRCUIT BREAKER CABINET LIGHTING / INPUT CABINET LIGHT CIRCUIT BREAKER TRIPPED
      INPUT_SENTRON_PAC_BREAKER : Bool;   // INPUT BREAKER SENTRON PAC3200 / INPUT SENTRON PAC CIRCUIT BREAKER TRIPPED
      INPUT_JIB_CRANE_BREAKER : Bool;   // CIRCUIT BREAKER JIB CRANE / INPUT JIB CRANE CIRCUIT BREAKER TRIPPED
      INPUT_MAIN_SWITCH : Bool;   // ELECTRICAL CABINET MAIN SWITCH INPUT / INPUT MAIN SWITCH
      INPUT_PANEL_TEMPERATURE : Bool;   // PANEL TEMPERATURE STOP END OF CYCLE / INPUT PANEL TEMPERATURE
      INPUT_AIR_UNIT_1 : Bool;   // AIR UNIT OK - STOP END OF CYCLE / INPUT AIR UNIT 1
      INPUT_AIR_UNIT_2 : Bool;   // AIR UNIT OK - STOP END OF CYCLE / INPUT AIR UNIT 2
      INPUT_OVER_VOLTAGE : Bool;   // INPUT OVER VOLTAGE
      INPUT_POWER_SUPPLY : Bool;   // FAULT POWER SUPPLY / INPUT POWER SUPPLY
      INPUT_PS_24V_NOT_READY_DEV_1 : Bool;   // INPUT POWER SUPPLY 24V NOT READY DEVICE 1
      INPUT_PS_24V_NOT_READY_DEV_2 : Bool;   // INPUT POWER SUPPLY 24V NOT READY DEVICE 2
      INPUT_PS_24V_NOT_READY_DEV_3 : Bool;   // INPUT POWER SUPPLY 24V NOT READY DEVICE 3
      INPUT_PS_24V_NOT_READY_DEV_4 : Bool;   // INPUT POWER SUPPLY 24V NOT READY DEVICE 4
      INPUT_PS_24V_NOT_READY_DEV_5 : Bool;   // INPUT POWER SUPPLY 24V NOT READY DEVICE 5
      INPUT_PS_24V_NOT_READY_DEV_6 : Bool;   // INPUT POWER SUPPLY 24V NOT READY DEVICE 6
      INPUT_BATTERY_OK_SITOP_UPS500S : Bool;   // INPUT BATTERY OK SITOP UPS500S
      INPUT_BATTERY_ALARM_SITOP_UPS500S : Bool;   // INPUT BATTERY ALARM SITOP UPS500S
      INPUT_ETHERNET_SWITCH_1 : Bool;   // INPUT SWITCH ETHERNET SWITCH 1 FAULT / INPUT ETHERNET SWITCH 1
      INPUT_ETHERNET_SWITCH_2 : Bool;   // INPUT SWITCH ETHERNET SWITCH 2 FAULT / INPUT ETHERNET SWITCH 2
      INPUT_ETHERNET_SWITCH_3 : Bool;   // INPUT SWITCH ETHERNET SWITCH 3 FAULT / INPUT ETHERNET SWITCH 3
      INPUT_ETHERNET_SWITCH_4 : Bool;   // INPUT ETHERNET SWITCH 4
      INPUT_ELEC_CAB_DOOR_OPEN : Bool;   // INPUT ELECTRICAL CABINET DOOR OPENED / INPUT ELECTRICAL CABINET DOOR OPEN
      INPUT_BATTERY_85_SITOP_UPS500S : Bool;   // INPUT BATTERY 85% SITOP UPS500S
      INPUT_PS_24V_BREAKER_DEV_1 : Bool;   // POWER SUPPLY 24V CIRCUIT BREAKER TRIPPED DEVICE 1 INPUT (WITHOUT FB) / INPUT POWER SUPPLY 24V CIRCUIT BREAKER TRIPPED DEVICE 1
      INPUT_PS_24V_BREAKER_DEV_2 : Bool;   // POWER SUPPLY 24V CIRCUIT BREAKER TRIPPED DEVICE 2 INPUT (WITHOUT FB) / INPUT POWER SUPPLY 24V CIRCUIT BREAKER TRIPPED DEVICE 2
      INPUT_PS_24V_BREAKER_DEV_3 : Bool;   // POWER SUPPLY 24V CIRCUIT BREAKER TRIPPED DEVICE 3 INPUT (WITHOUT FB) / INPUT POWER SUPPLY 24V CIRCUIT BREAKER TRIPPED DEVICE 3
      INPUT_PS_24V_BREAKER_DEV_4 : Bool;   // POWER SUPPLY 24V CIRCUIT BREAKER TRIPPED DEVICE 4 INPUT (WITHOUT FB) / INPUT POWER SUPPLY 24V CIRCUIT BREAKER TRIPPED DEVICE 4
      INPUT_LASER_BREAKER_U01 : Bool;   // INPUT LASER SOURCE UNIT 01 CIRCUIT BREAKER TRIPPED
      INPUT_LASER_BREAKER_U02 : Bool;   // INPUT LASER SOURCE UNIT 02 CIRCUIT BREAKER TRIPPED
      INPUT_OERLIKON_BREAKER_U01 : Bool;   // INPUT OERLIKON SOURCE UNIT 01 CIRCUIT BREAKER TRIPPED
      INPUT_OERLIKON_BREAKER_U02 : Bool;   // INPUT OERLIKON SOURCE UNIT 02 CIRCUIT BREAKER TRIPPED
      INPUT_HEATER_BREAKER : Bool;   // INPUT HEATER CIRCUIT BREAKER TRIPPED
      INPUT_AXIS_Z11_BREAKER_1 : Bool;   // INPUT AXIS Z11 CIRCUIT BREAKER 1 TRIPPED
      INPUT_AXIS_Z11_BREAKER_2 : Bool;   // INPUT AXIS Z11 CIRCUIT BREAKER 2 TRIPPED
      INPUT_STIRRER_BREAKER : Bool;   // INPUT STIRRER CIRCUIT BREAKER 2 TRIPPED
      INPUT_CHILLER_BREAKER_1 : Bool;   // INPUT CHILLER CIRCUIT BREAKER 2 TRIPPED
      INPUT_HOPPERS_BREAKER : Bool;   // INPUT HOPPERS CIRCUIT BREAKER 2 TRIPPED
      INPUT_AXIS_Z21_BREAKER_1 : Bool;   // INPUT AXIS Z21 CIRCUIT BREAKER 1 TRIPPED
      INPUT_AXIS_Z21_BREAKER_2 : Bool;   // INPUT AXIS Z21 CIRCUIT BREAKER 2 TRIPPED
      "230_VAC_BREAKER_TRIPPED_ALARM" : Bool;   // MAIN CIRCUIT BREAKER FAULT / 230 VAC BREAKER TRIPPED ALARM
      INPUT_PILZ_ESTOP_OK : Bool;   // INPUT PILZ EMERGENCY STOP OK
      AIR_UNIT_1_BREAKER_TRIPPED_ALARM : Bool;   // AIR UNIT CIRCUIT BREAKER FAULT / AIR UNIT 1 CIRCUIT BREAKER TRIPPED ALARM
      AIR_UNIT_2_BREAKER_TRIPPED_ALARM : Bool;   // AIR UNIT CIRCUIT BREAKER FAULT / AIR UNIT 2 CIRCUIT BREAKER TRIPPED ALARM
      "24VDC_BREAKER_TRIPPED_ALARM_1" : Bool;   // CIRCUIT BREAKER 24 V DC FAULT / 24 VDC CIRCUIT BREAKER TRIPPED 1 ALARM
      "24VDC_BREAKER_TRIPPED_ALARM_2" : Bool;   // AUXILIAR CIRCUIT BRAKER 24 VDC FAULT / 24 VDC CIRCUIT BREAKER TRIPPED 2 ALARM
      FC35_1_BREAKER_TRIPPED_ALARM : Bool;   // BREAKER QF3004 FAULT / FC35.1 CIRCUIT BREAKER TRIPPED ALARM
      FC35_2_BREAKER_TRIPPED_ALARM : Bool;   // BREAKER QF3004 FAULT / FC35.2 CIRCUIT BREAKER TRIPPED ALARM
      FC35_3_BREAKER_TRIPPED_ALARM : Bool;   // BREAKER QF3004 FAULT / FC35.3 CIRCUIT BREAKER TRIPPED ALARM
      SINAMICS_BREAKER_TRIPPED_ALARM : Bool;   // SINAMICS CIRCUIT BREAKER TRIPPED FAULT / SINAMICS CIRCUIT BREAKER TRIPPED ALARM
      MAIN_SWITCH_ALARM : Bool;   // MAIN SWITCH OFF FAULT / MAIN SWITCH ALARM
      PANEL_TEMPERATURE_ALARM : Bool;   // PANEL TEMPERATURE NOT OK - STOP END OF CYCLE / PANEL TEMPERATURE ALARM
      AIR_UNIT_ALARM_1 : Bool;   // AIR UNIT NOT OK - STOP END OF CYCLE / AIR UNIT 1 ALARM
      AIR_UNIT_ALARM_2 : Bool;   // AIR UNIT NOT OK - STOP END OF CYCLE / AIR UNIT 2 ALARM
      OVER_VOLTAGE_ALARM : Bool;   // OVER VOLTAGE FAULT / OVER VOLTAGE ALARM
      POWER_SUPPLY_ALARM : Bool;   // POWER SUPPLY FAULT / POWER SUPPLY ALARM
      PS_24V_NOT_READY_DEV_ALARM_1 : Bool;   // POWER SUPPLY 24V NOT READY DEVICE 1 ALARM
      PS_24V_NOT_READY_DEV_ALARM_2 : Bool;   // POWER SUPPLY 24V NOT READY DEVICE 2 ALARM
      PS_24V_NOT_READY_DEV_ALARM_3 : Bool;   // POWER SUPPLY 24V NOT READY DEVICE 3 ALARM
      PS_24V_NOT_READY_DEV_ALARM_4 : Bool;   // POWER SUPPLY 24V NOT READY DEVICE 4 ALARM
      PS_24V_NOT_READY_DEV_ALARM_5 : Bool;   // POWER SUPPLY 24V NOT READY DEVICE 5 ALARM
      PS_24V_NOT_READY_DEV_ALARM_6 : Bool;   // POWER SUPPLY 24V NOT READY DEVICE 6 ALARM
      BATTERY_OK_SITOP_UPS500S_ALARM : Bool;   // SITOP UPS500S BATTERY NOT OK ALARM / BATTERY OK SITOP UPS500S ALARM
      BATTERY_ALARM_SITOP_UPS500S : Bool;   // SITOP UPS500S BATTERY LOW LEVEL ALARM / BATTERY ALARM SITOP UPS500S ALARM
      ETHERNET_SWITCH_1_ALARM : Bool;   // SWITCH SCALANCE X108 FAIL / ETHERNET SWITCH 1 ALARM
      ETHERNET_SWITCH_2_ALARM : Bool;   // ETHERNET SWITCH 2 ALARM
      ETHERNET_SWITCH_3_ALARM : Bool;   // ETHERNET SWITCH 3 ALARM
      ETHERNET_SWITCH_4_ALARM : Bool;   // ETHERNET SWITCH 4 ALARM
      PS_24V_BREAKER_TRIPPED_ALARM_DEV_1 : Bool;   // DIAGNOSIS 24V MODULE CIRCUIT BREAKER 1 TRIPPED / POWER SUPPLY 24V CIRCUIT BREAKER TRIPPED DEVICE 1 ALARM
      PS_24V_BREAKER_TRIPPED_ALARM_DEV_2 : Bool;   // DIAGNOSIS 24V MODULE CIRCUIT BREAKER 2 TRIPPED / POWER SUPPLY 24V CIRCUIT BREAKER TRIPPED DEVICE 2 ALARM
      PS_24V_BREAKER_TRIPPED_ALARM_DEV_3 : Bool;   // DIAGNOSIS 24V MODULE CIRCUIT BREAKER 3 TRIPPED / POWER SUPPLY 24V CIRCUIT BREAKER TRIPPED DEVICE 3 ALARM
      PS_24V_BREAKER_TRIPPED_ALARM_DEV_4 : Bool;   // DIAGNOSIS 24V MODULE CIRCUIT BREAKER 4 TRIPPED / POWER SUPPLY 24V CIRCUIT BREAKER TRIPPED DEVICE 4 ALARM
      SINAMICS_BREAKER_ALARM : Bool;   // SINAMICS CIRCUIT BREAKER TRIPPED ALARM
      LASER_BREAKER_U01_ALARM : Bool;   // ALARM LASER SOURCE UNIT 01 CIRCUIT BREAKER TRIPPED
      LASER_BREAKER_U02_ALARM : Bool;   // ALARM LASER SOURCE UNIT 02 CIRCUIT BREAKER TRIPPED
      OERLIKON_BREAKER_U01_ALARM : Bool;   // ALARM OERLIKON SOURCE UNIT 01 CIRCUIT BREAKER TRIPPED
      OERLIKON_BREAKER_U02_ALARM : Bool;   // ALARM OERLIKON SOURCE UNIT 02 CIRCUIT BREAKER TRIPPED
      HEATER_BREAKER_ALARM : Bool;   // ALARM HEATER CIRCUIT BREAKER TRIPPED
      AXIS_Z11_BREAKER_1_ALARM : Bool;   // ALARM AXIS Z11 CIRCUIT BREAKER 1 TRIPPED
      AXIS_Z11_BREAKER_2_ALARM : Bool;   // ALARM AXIS Z11 CIRCUIT BREAKER 2 TRIPPED
      STIRRER_BREAKER_ALARM : Bool;   // ALARM STIRRER CIRCUIT BREAKER TRIPPED
      CHILLER_BREAKER_ALARM : Bool;   // ALARM CHILLER CIRCUIT BREAKER TRIPPED
      HOPPERS_BREAKER_ALARM : Bool;   // ALARM HOPPERS CIRCUIT BREAKER TRIPPED
      AXIS_Z21_BREAKER_1_ALARM : Bool;   // ALARM AXIS Z21 CIRCUIT BREAKER 1 TRIPPED
      AXIS_Z21_BREAKER_2_ALARM : Bool;   // ALARM AXIS Z21 CIRCUIT BREAKER 2 TRIPPED
      "110/120/220/230VAC_BREAKER_TRIPPED_WARNING" : Bool;   // BREAKER 120VA TRIPPED / 110/120/220/230VAC CIRCUIT BREAKER TRIPPED WARNING
      CAB_LIGHT_BREAKER_TRIPPED_WARNING : Bool;   // CIRCUIT BREAKER CABINET LIGHTING WARNING / CABINET LIGHT CIRCUIT BREAKER TRIPPED WARNING
      SENTRON_PAC_BREAKER_TRIPPED_WARNING : Bool;   // CIRCUIT BREAKER SENTRON PACK3200 TRIPPED / SENTRON PAC CIRCUIT BREAKER TRIPPED WARNING
      JIB_CRANE_BREAKER_TRIPPED_WARNING : Bool;   // CIRCUIT BREAKER JIB CRANE FAULT / JIB CRANE CIRCUIT BREAKER TRIPPED WARNING
      ELEC_CAB_DOOR_OPEN_WARNING : Bool;   // ELECTRICAL CABINET DOOR OPENED / ELECTRICAL CABINET DOOR OPEN WARNING
      BATTERY_85_SITOP_UPS500S_WARNING : Bool;   // SITOP UPS500S BATTERY 85 WARNING / BATTERY 85% SITOP UPS500S WARNING
      PILZ_ESTOP_OK_ALARM : Bool;   // PILZ EMERGENCY STOP OK ALARM
      ANY_ACTIVE_ALARM : Bool;   // RETURN TO HOME POSITION ALARMS / ANY ACTIVE ALARM
      IS_ALARMS : Bool;   // IMMEDIATE STOP ALARMS
      SEOC_ALARMS : Bool;   // STOP AT END OF CYCLE ALARMS / STOP END OF CYCLE ALARMS
      WARNINGS : Bool;   // WARNING / WARNINGS
      WARNINGS_GONE : Bool;   // WARNING GONE / WARNINGS GONE
      TIMER_SITOP_BATTERY { S7_SetPoint := 'True'} : TON_TIME;   // SITOP BATTERY TIMER
   END_VAR
BEGIN
   TIMER_SITOP_BATTERY.PT := T#5s;
END_DATA_BLOCK

DATA_BLOCK "DB2107_MACHINE_LIGHT"   // DB2107
{ S7_Optimized_Access := 'FALSE'; DB_Accessible_From_OPC_UA := 'FALSE' }
AUTHOR : ETXETAR
VERSION : 1.0
// stored: AutoNumber false, DBAccessibleFromOPCUA false, DBAccessibleFromWebserver true, IsOnlyStoredInLoadMemory false, IsWriteProtectedInAS false
   VAR RETAIN
      I_CIRCUIT_BREAKER : Bool;   // CIRCUIT BREAKER INPUT
      I_SELECTOR_ON : Bool;   // SELECTOR ON INPUT
      SWITCH_ON_GENERAL_CONDITIONS : Bool;   // SWITCH ON GENERAL CONDITIONS
      SWITCH_ON_INITIAL_CONDITIONS : Bool;   // SWITCH ON INITIAL CONDITIONS
      SWITCH_ON_MANUAL_REQUEST : Bool;   // SWITCH ON MANUAL REQUEST
      SWITCH_ON_AUTO_REQUEST : Bool;   // SWITCH ON AUTO REQUEST
      SWITCH_ON_GLOBAL_REQUEST : Bool;   // SWITCH ON GLOBAL REQUEST
      SWITCH_ON_COMMAND : Bool;   // SWITCH ON COMMAND
      SWITCH_ON : Bool;   // SWITCH ON
      IN_SERVICE : Bool;   // IN SERVICE
      SWITCH_OFF_GENERAL_CONDITIONS : Bool;   // SWITCH OFF GENERAL CONDITIONS
      SWITCH_OFF_INITIAL_CONDITIONS : Bool;   // SWITCH OFF INITIAL CONDITIONS
      SWITCH_OFF_MANUAL_REQUEST : Bool;   // SWITCH OFF MANUAL REQUEST
      SWITCH_OFF_AUTO_REQUEST : Bool;   // SWITCH OFF AUTO REQUEST
      SWITCH_OFF_GLOBAL_REQUEST : Bool;   // SWITCH OFF GLOBAL REQUEST
      SWITCH_OFF_COMMAND : Bool;   // SWITCH OFF COMMAND
      SWITCH_OFF : Bool;   // SWITCH OFF
      OUT_OF_SERVICE : Bool;   // OUT OF SERVICE
      SWITCH_ON_GENERAL_CONDITIONS_HELP : Bool;   // SWITCH ON GENERAL CONDITIONS HELP
      SWITCH_ON_INITIAL_CONDITIONS_HELP : Bool;   // SWITCH ON INITIAL CONDITIONS HELP
      SWITCH_OFF_GENERAL_CONDITIONS_HELP : Bool;   // SWITCH OFF GENERAL CONDITIONS HELP
      SWITCH_OFF_INITIAL_CONDITIONS_HELP : Bool;   // SWITCH OFF INITIAL CONDITIONS HELP
      SWITCH_ON_GLOBAL_REQUEST_AUX1 : Bool;   // SWITCH ON GLOBAL REQUEST ON AUXILIARY 1
      SWITCH_ON_GLOBAL_REQUEST_AUX2 : Bool;   // SWITCH ON GLOBAL REQUEST ON AUXILIARY 2
      SWITCH_ON_GLOBAL_REQUEST_AUX3 : Bool;   // SWITCH ON GLOBAL REQUEST ON AUXILIARY 3
      SWITCH_OFF_AUTO_REQUEST_AUX : Bool;   // INITIAL AUX 4
      SWITCH_OFF_GLOBAL_REQUEST_AUX : Bool;   // INITIAL AUX 5
      TIMER_SWITCH_OFF_1 : TON_TIME;   // SWITCH OFF GLOBAL REQUEST 1 TIMER
      TIMER_SWITCH_OFF_2 : TON_TIME;   // SWITCH OFF GLOBAL REQUEST 2 TIMER
   END_VAR
BEGIN
   TIMER_SWITCH_OFF_1.PT := T#10M;
   TIMER_SWITCH_OFF_2.PT := T#1H;
END_DATA_BLOCK

DATA_BLOCK "DB2120_MPP_ITC_IPC"   // DB2120
{ S7_Optimized_Access := 'FALSE'; DB_Accessible_From_OPC_UA := 'FALSE' }
AUTHOR : ETXETAR
VERSION : 1.0
// stored: AutoNumber false, DBAccessibleFromOPCUA false, DBAccessibleFromWebserver true, IsOnlyStoredInLoadMemory false, IsWriteProtectedInAS false
   VAR RETAIN
      INPUT_CONTROL_ON : Bool;   // INPUT CONTROL ON
      CONTROL_ON : Bool;   // CONTROL ON
      CONTROL_ON_DELAYED : Bool;   // CONTROL ON DELAYED
      CONTROL_ON_PULSE : Bool;   // CONTROL ON PULSE
      CONTROL_OFF3_DELAYED : Bool;   // MACHINE OFF DELAYED / CONTROL OFF3 DELAYED
      CONTROL_ON_OFF_DELAYED : Bool;   // MACHINE OFF DELAYED / CONTROL ON/OFF DELAYED
      MACHINE_ON : Bool;   // MACHINE ON
      MACHINE_ON_DELAYED : Bool;   // MACHINE ON DELAYED
      MACHINE_OFF_DELAYED : Bool;   // MACHINE OFF DELAYED
      MACHINE_ON_DELAYED_PULSE : Bool;   // MACHINE ON DELAYED PULSE
      MACHINE_ON_DELAYED_AUX : Bool;   // MACHINE ON DELAYED AUXILIARY
      MACH_ON_DEL_PNEU_ON : Bool;   // CRM + HYD + PNEUMATIC ON / MACHINE ON DELAYED PNEUMATIC IN SERVICE
      MACH_STOP_SERV_ENABLED : Bool;   // MACHINE STOP SERVICES DELAYED ENABLED
      MACH_STOP_SERV_DELAY_1 : Bool;   // MACHINE STOP SERVICES DELAYED 1
      MACH_STOP_SERV_DELAY_2 : Bool;   // MACHINE STOP SERVICES DELAYED 2
      MPP_MAIN_PANEL_ACTIVE : Bool;   // MPP MAIN PANEL ACTIVE
      ITC_1_ACTIVE : Bool;   // TCU 1 ACTIVE / ITC 1 ACTIVE
      HT10_ACTIVE : Bool;   // HT8 ACTIVE / HT10 ACTIVE
      AXES_OVERRIDE : Byte;   // AXES OVERRIDE
      AXES_OVERRIDE_DECIMAL : Byte;   // RESERVED / AXES OVERRIDE VALUE IN DECIMAL
      SPINDLES_OVERRIDE : Byte;   // SPINDLES OVERRIDE
      OVERRIDE_ZERO : Bool;   // OVERRIDE ZERO
      OVERRIDE_LOWER_THAN_80 : Bool;   // OVERRIDE LOWER THAN 80
      OVERRIDE_100 : Bool;   // OVERRIDE 100
      START_SERVICES_GLOBAL : Bool;   // START SERVICES GLOBAL
      START_CYCLE_GLOBAL : Bool;   // START CYCLE GLOBAL
      RETURN_HOME_POSITION_BY_OPERATOR : Bool;   // RETURN HOME POSITION BY OPERATOR
      RETURN_HOME_POSITION_BY_OPERATOR_AUX_1 : Bool;   // RETURN HOME POSITION BY OPERATOR / RETURN HOME POSITION BY OPERATOR AUXILIARY 1
      RETURN_HOME_POSITION_BY_OPERATOR_AUX_2 : Bool;   // RETURN HOME POSITION BY OPERATOR / RETURN HOME POSITION BY OPERATOR AUXILIARY 2
      RETURN_HOME_POSITION_FROM_MPP_PANEL : Bool;   // RETURN HOME POSITION FROM MPP PANNEL / RETURN HOME POSITION FROM MPP PANEL
      RETURN_HOME_POSITION_FROM_AUX_PANEL : Bool;   // RETURN HOME POSITION FROM AUX PANEL
      RETURN_HOME_POSITION_PULSE : Bool;   // END OF CYCLE TOGGLE AUXILIAR FUNCTION / RETURN HOME POSITION PULSE
      RESET_FAULTS : Bool;   // RESET FAULT / RESET FAULTS
      RESET_FAULTS_PULSE : Bool;   // RESET FAULT PULSE / RESET FAULTS PULSE
      RESET_FAULTS_GLOBAL : Bool;   // RESET FAULTS GLOBAL
      RESET_FAULTS_AUX : Bool;   // AUXILIARY RESET FAULT / RESET FAULTS AUXILIARY
      STOP_SERVICES_GLOBAL : Bool;   // STOP SERVICES GLOBAL
      STOP_END_OF_CYCLE_REQUEST : Bool;   // STOP END OF CYCLE REQUEST
      AUX_STOP_END_CYCLE_REQUEST : Bool;   // AUX STOP END CYCLE REQUEST
      STOP_END_OF_CYCLE_FROM_MPP_PANEL : Bool;   // END OF CYCLE FROM MPP PANNEL / STOP END OF CYCLE FROM MPP PANEL
      STOP_END_OF_CYCLE_FROM_AUX_PANEL : Bool;   // END OF CYCLE FROM AUX PANNEL / STOP END OF CYCLE FROM AUX PANEL
      STOP_END_OF_CYCLE_BY_OPERATOR : Bool;   // STOP END OF CYCLE BY OPERATOR
      STOP_END_OF_CYCLE_BY_OPERATOR_AUX_1 : Bool;   // STOP END OF CYCLE BY OPERATOR / STOP END OF CYCLE BY OPERATOR AUXILIARY 1
      STOP_END_OF_CYCLE_BY_OPERATOR_AUX_2 : Bool;   // STOP END OF CYCLE BY OPERATOR / STOP END OF CYCLE BY OPERATOR AUXILIARY 2
      STOP_END_OF_CYCLE_PULSE : Bool;   // END OF CYCLE BY OPERATOR ACTIVE / STOP END OF CYCLE PULSE
      IMMEDIATE_STOP_BY_OPERATOR : Bool;   // IMMEDIATY STOP BY OPERATOR / IMMEDIATE STOP BY OPERATOR
      IMMEDIATE_STOP_BY_OPERATOR_AUX : Bool;   // IMMEDIATY STOP BY OPERATOR / IMMEDIATE STOP BY OPERATOR AUXILIARY
      IMMEDIATE_STOP_GLOBAL : Bool;   // IMMEDIATE STOP GLOBAL
      SAFETY_DOORS_NOT_CLOSED : Bool;   // PILZS GATES NOT CLOSED / SAFETY DOORS NOT CLOSED
      ANY_SAFETY_DOOR_UNLOCK_COMAND : Bool;   // ANY SAFETY DOOR UNLOCK COMMAND
      ANY_SAFETY_DOOR_UNLOCK : Bool;   // ANY SAFETY DOOR UNLOCK
      BIMANUAL_F1_UNLOAD_PARTS_CONDITIONS : Bool;   // BIMANUAL FIXTURE 1 UNLOAD PARTS CONDITIONS
      BIMANUAL_F2_UNLOAD_PARTS_CONDITIONS : Bool;   // BIMANUAL FIXTURE 2 UNLOAD PARTS CONDITIONS
      TIMER_CONTROL_ON : TON_TIME;   // CONTROL ON TIMER
      TIMER_MACHINE_ON : TON_TIME;   // MACHINE ON TIMER
      TIMER_MACHINE_OFF : TOF_TIME;   // MACHINE OFF TIMER
      TIMER_MACH_STOP_SERV_DELAY : TON_TIME;   // MACHINE STOP SERVICES TIMER
      TIMER_BIMANUAL_CYCLE_START : TON_TIME;   // BIMANUAL CYCLE START TIMER
      TIMER_CONTROL_OFF : TOF_TIME;   // CONTROL OFF TIMER
      TIMER_CONTROL_OFF3 : TOF_TIME;   // CONTROL OFF3 TIMER
      TIMER_CONTROL_ON_OFF : TOF_TIME;   // CONTROL ON/OFF TIMER
   END_VAR
BEGIN
   TIMER_CONTROL_ON.PT := T#3s;
   TIMER_MACHINE_ON.PT := T#2s;
   TIMER_MACHINE_OFF.PT := T#3s;
   TIMER_BIMANUAL_CYCLE_START.PT := T#2s;
   TIMER_CONTROL_OFF.PT := T#1s;
   TIMER_CONTROL_OFF3.PT := T#5s;
   TIMER_CONTROL_ON_OFF.PT := T#6s;
END_DATA_BLOCK

DATA_BLOCK "DB2121_MPP"   // DB2121
{ S7_Optimized_Access := 'FALSE'; DB_Accessible_From_OPC_UA := 'FALSE' }
AUTHOR : ETXETAR
VERSION : 1.0
// stored: AutoNumber false, DBAccessibleFromOPCUA false, DBAccessibleFromWebserver true, IsOnlyStoredInLoadMemory false, IsWriteProtectedInAS false
   VAR
      INPUTS : "MPP_INPUTS";
      OUTPUTS : "MPP_OUTPUTS";
      OVERRIDE_AUX : Struct
         FEED_OVERRIDE : Struct
            I_WS2_1_FEED_OVERRIDE : Bool;   // WS2/1 - FEEDRATE OVERRIDE
            I_WS2_2_FEED_OVERRIDE : Bool;   // WS2/2 - FEEDRATE OVERRIDE
            I_WS2_4_FEED_OVERRIDE : Bool;   // WS2/4 - FEEDRATE OVERRIDE
            I_WS2_8_FEED_OVERRIDE : Bool;   // WS2/8 - FEEDRATE OVERRIDE
            I_WS2_16_FEED_OVERRIDE : Bool;   // WS2/16 - FEEDRATE OVERRIDE
            I_28_5 : Bool;   // NOT USED
            I_28_6 : Bool;   // NOT USED
            I_28_7 : Bool;   // NOT USED
         END_STRUCT;
         SPINDLES_OVERRIDE : Struct
            I_WS3_1_SPIND_OVERRIDE : Bool;   // WS3/1 - SPINDLE OVERRIDE
            I_WS3_2_SPIND_OVERRIDE : Bool;   // WS3/2 - SPINDLE OVERRIDE
            I_WS3_4_SPIND_OVERRIDE : Bool;   // WS3/4 - SPINDLE OVERRIDE
            I_WS3_8_SPIND_OVERRIDE : Bool;   // WS3/8 - SPINDLE OVERRIDE
            I_WS3_16_SPIND_OVERRIDE : Bool;   // WS3/16 - SPINDLE OVERRIDE
            I_30_5 : Bool;   // NOT USED
            I_30_6 : Bool;   // NOT USED
            I_30_7 : Bool;   // NOT USED
         END_STRUCT;
      END_STRUCT;
      INPUT_PANEL_EMERGENCY_STOP : Bool;   // INPUT PANEL EMERGENCY STOP
      INPUT_BYPASS_SAFETY_DOOR : Bool;   // INPUT BYPASS SAFETY DOOR
      EMERGENCY_STOP_ACTIVE : Bool;   // EMERGENCY STOP ACTIVE PILZ / EMERGENCY STOP ACTIVE
      BYPASS_SAFETY_DOOR_ACTIVE : Bool;   // BYPASS SAFETY DOOR ACTIVE
      NEXT_AXES_RQ_CND : Bool;   // NEXT AXES REQUEST CONDITIONS
      NEXT_AXES_SELECT_RST : Bool;   // NEXT AXES SELECT RESET
      NEXT_AXES_SELECT_CMM_P : Bool;   // NEXT AXES SELECT COMMAND PULSE
      NEXT_AXES_SELECT_AUX : Bool;   // NEXT AXES SELECT AUXILIARY
      NEXT_AXES_RQ_P : Bool;   // NEXT AXES REQUEST PULSE
      NEXT_AXES_ANY_AX_RQ : Bool;   // NEXT AXES ANY AXIS REQUEST
      PULSE : Bool;   // PULSE
      PULSE1 : Bool;   // PULSE 1
      PULSE2 : Bool;   // PULSE 2
      TIMER_NEXT_AXES_1 : TON_TIME;
      TIMER_NEXT_AXES_2 : TON_TIME;
   END_VAR
BEGIN
   TIMER_NEXT_AXES_1.PT := T#500ms;
   TIMER_NEXT_AXES_2.PT := T#500ms;
END_DATA_BLOCK

DATA_BLOCK "DB2122_HT10"   // DB2122
{ S7_Optimized_Access := 'FALSE'; DB_Accessible_From_OPC_UA := 'FALSE' }
AUTHOR : ETXETAR
VERSION : 1.0
// stored: AutoNumber false, DBAccessibleFromOPCUA false, DBAccessibleFromWebserver true, IsOnlyStoredInLoadMemory false, IsWriteProtectedInAS false
   VAR
      INPUT_HT10_EMERGENCY_STOP : Bool;   // INPUT HT8 EMERGENCY STOP / INPUT HT10 EMERGENCY STOP
      HT10_EMERGENCY_STOP_ACTIVE : Bool;   // HT8 EMERGENCY STOP ACTIVE / HT10 EMERGENCY STOP ACTIVE
      INPUTS : "HT10_INPUTS";   // HT10 INPUTS
      ENABLE_CHANGE { S7_SetPoint := 'True'} : "HT10_ENABLE_CHANGE";
   END_VAR
BEGIN
END_DATA_BLOCK

DATA_BLOCK "DB2140_HOPPERS_MPP"   // DB2140
{ S7_Optimized_Access := 'FALSE'; DB_Accessible_From_OPC_UA := 'FALSE' }
AUTHOR : ETXETAR
VERSION : 1.0
// stored: AutoNumber false, DBAccessibleFromOPCUA false, DBAccessibleFromWebserver true, IsOnlyStoredInLoadMemory false, IsWriteProtectedInAS false
   VAR RETAIN
      INPUT_CONTROL_ON : Bool;   // INPUT CONTROL ON
      INPUT_CONTROL_OFF : Bool;   // INPUT CONTROL OFF
      CONTROL_ON : Bool;   // CONTROL ON
      CONTROL_ON_DELAYED : Bool;   // CONTROL ON DELAYED
      CONTROL_ON_PULSE : Bool;   // CONTROL ON PULSE
      CONTROL_OFF3_DELAYED : Bool;   // MACHINE OFF DELAYED / CONTROL OFF3 DELAYED
      CONTROL_ON_OFF_DELAYED : Bool;   // MACHINE OFF DELAYED / CONTROL ON/OFF DELAYED
      MACHINE_ON : Bool;   // MACHINE ON
      MACHINE_ON_DELAYED : Bool;   // MACHINE ON DELAYED
      MACHINE_OFF_DELAYED : Bool;   // MACHINE OFF DELAYED
      MACHINE_ON_DELAYED_PULSE : Bool;   // MACHINE ON DELAYED PULSE
      MACHINE_ON_DELAYED_AUX : Bool;   // MACHINE ON DELAYED AUXILIARY
      MACH_ON_DEL_PNEU_ON : Bool;   // CRM + HYD + PNEUMATIC ON / MACHINE ON DELAYED PNEUMATIC IN SERVICE
      MACH_STOP_SERV_ENABLED : Bool;   // MACHINE STOP SERVICES DELAYED ENABLED
      MACH_STOP_SERV_DELAY_1 : Bool;   // MACHINE STOP SERVICES DELAYED 1
      MACH_STOP_SERV_DELAY_2 : Bool;   // MACHINE STOP SERVICES DELAYED 2
      MPP_MAIN_PANEL_ACTIVE : Bool;   // MPP MAIN PANEL ACTIVE
      ITC_1_ACTIVE : Bool;   // TCU 1 ACTIVE / ITC 1 ACTIVE
      HT10_ACTIVE : Bool;   // HT8 ACTIVE / HT10 ACTIVE
      AXES_OVERRIDE : Byte;   // AXES OVERRIDE
      AXES_OVERRIDE_DECIMAL : Byte;   // RESERVED / AXES OVERRIDE VALUE IN DECIMAL
      SPINDLES_OVERRIDE : Byte;   // SPINDLES OVERRIDE
      OVERRIDE_ZERO : Bool;   // OVERRIDE ZERO
      OVERRIDE_LOWER_THAN_80 : Bool;   // OVERRIDE LOWER THAN 80
      OVERRIDE_100 : Bool;   // OVERRIDE 100
      START_SERVICES_GLOBAL : Bool;   // START SERVICES GLOBAL
      START_CYCLE_GLOBAL : Bool;   // START CYCLE GLOBAL
      RETURN_HOME_POSITION_BY_OPERATOR : Bool;   // RETURN HOME POSITION BY OPERATOR
      RETURN_HOME_POSITION_BY_OPERATOR_AUX_1 : Bool;   // RETURN HOME POSITION BY OPERATOR / RETURN HOME POSITION BY OPERATOR AUXILIARY 1
      RETURN_HOME_POSITION_BY_OPERATOR_AUX_2 : Bool;   // RETURN HOME POSITION BY OPERATOR / RETURN HOME POSITION BY OPERATOR AUXILIARY 2
      RETURN_HOME_POSITION_FROM_MPP_PANEL : Bool;   // RETURN HOME POSITION FROM MPP PANNEL / RETURN HOME POSITION FROM MPP PANEL
      RETURN_HOME_POSITION_FROM_AUX_PANEL : Bool;   // RETURN HOME POSITION FROM AUX PANEL
      RETURN_HOME_POSITION_PULSE : Bool;   // END OF CYCLE TOGGLE AUXILIAR FUNCTION / RETURN HOME POSITION PULSE
      RESET_FAULTS : Bool;   // RESET FAULT / RESET FAULTS
      RESET_FAULTS_PULSE : Bool;   // RESET FAULT PULSE / RESET FAULTS PULSE
      RESET_FAULTS_GLOBAL : Bool;   // RESET FAULTS GLOBAL
      RESET_FAULTS_AUX : Bool;   // AUXILIARY RESET FAULT / RESET FAULTS AUXILIARY
      STOP_SERVICES_GLOBAL : Bool;   // STOP SERVICES GLOBAL
      STOP_END_OF_CYCLE_REQUEST : Bool;   // STOP END OF CYCLE REQUEST
      AUX_STOP_END_CYCLE_REQUEST : Bool;   // AUX STOP END CYCLE REQUEST
      STOP_END_OF_CYCLE_FROM_MPP_PANEL : Bool;   // END OF CYCLE FROM MPP PANNEL / STOP END OF CYCLE FROM MPP PANEL
      STOP_END_OF_CYCLE_FROM_AUX_PANEL : Bool;   // END OF CYCLE FROM AUX PANNEL / STOP END OF CYCLE FROM AUX PANEL
      STOP_END_OF_CYCLE_BY_OPERATOR : Bool;   // STOP END OF CYCLE BY OPERATOR
      STOP_END_OF_CYCLE_BY_OPERATOR_AUX_1 : Bool;   // STOP END OF CYCLE BY OPERATOR / STOP END OF CYCLE BY OPERATOR AUXILIARY 1
      STOP_END_OF_CYCLE_BY_OPERATOR_AUX_2 : Bool;   // STOP END OF CYCLE BY OPERATOR / STOP END OF CYCLE BY OPERATOR AUXILIARY 2
      STOP_END_OF_CYCLE_PULSE : Bool;   // END OF CYCLE BY OPERATOR ACTIVE / STOP END OF CYCLE PULSE
      IMMEDIATE_STOP_BY_OPERATOR : Bool;   // IMMEDIATY STOP BY OPERATOR / IMMEDIATE STOP BY OPERATOR
      IMMEDIATE_STOP_BY_OPERATOR_AUX : Bool;   // IMMEDIATY STOP BY OPERATOR / IMMEDIATE STOP BY OPERATOR AUXILIARY
      IMMEDIATE_STOP_GLOBAL : Bool;   // IMMEDIATE STOP GLOBAL
      SAFETY_DOORS_NOT_CLOSED : Bool;   // PILZS GATES NOT CLOSED / SAFETY DOORS NOT CLOSED
      ANY_SAFETY_DOOR_UNLOCK_COMAND : Bool;   // ANY SAFETY DOOR UNLOCK COMMAND
      ANY_SAFETY_DOOR_UNLOCK : Bool;   // ANY SAFETY DOOR UNLOCK
      BIMANUAL_F1_UNLOAD_PARTS_CONDITIONS : Bool;   // BIMANUAL FIXTURE 1 UNLOAD PARTS CONDITIONS
      BIMANUAL_F2_UNLOAD_PARTS_CONDITIONS : Bool;   // BIMANUAL FIXTURE 2 UNLOAD PARTS CONDITIONS
      IMMEDIATE_STOP_PULSE : Bool;   // INMEDIATE STOP PULSE
      TIMER_CONTROL_ON : TON_TIME;   // CONTROL ON TIMER
      TIMER_MACHINE_ON : TON_TIME;   // MACHINE ON TIMER
      TIMER_MACHINE_OFF : TOF_TIME;   // MACHINE OFF TIMER
      TIMER_MACH_STOP_SERV_DELAY : TON_TIME;   // MACHINE STOP SERVICES TIMER
      TIMER_BIMANUAL_CYCLE_START : TON_TIME;   // BIMANUAL CYCLE START TIMER
      TIMER_CONTROL_OFF : TOF_TIME;   // CONTROL OFF TIMER
      TIMER_CONTROL_OFF3 : TOF_TIME;   // CONTROL OFF3 TIMER
      TIMER_CONTROL_ON_OFF : TOF_TIME;   // CONTROL ON/OFF TIMER
   END_VAR
BEGIN
   TIMER_CONTROL_ON.PT := T#3s;
   TIMER_MACHINE_ON.PT := T#2s;
   TIMER_MACHINE_OFF.PT := T#3s;
   TIMER_BIMANUAL_CYCLE_START.PT := T#2s;
   TIMER_CONTROL_OFF.PT := T#1s;
   TIMER_CONTROL_OFF3.PT := T#5s;
   TIMER_CONTROL_ON_OFF.PT := T#6s;
END_DATA_BLOCK

DATA_BLOCK "DB2141_HOPPER_UNIT_01_IN_OUT"   // DB2141
{ S7_Optimized_Access := 'FALSE'; DB_Accessible_From_OPC_UA := 'FALSE' }
AUTHOR : ETXETAR
VERSION : 1.0
// stored: AutoNumber false, DBAccessibleFromOPCUA false, DBAccessibleFromWebserver true, IsOnlyStoredInLoadMemory false, IsWriteProtectedInAS false
   VAR
      BUTTONS : Struct
         CONTROL_ON : Bool;
         CONTROL_OFF : Bool;
         HOME_POSITION : Bool;
         AUTOMATIC_MODE : Bool;
         SEMIAUTOMATIC_MODE : Bool;
         MANUAL_MODE : Bool;
         START : Bool;
         STOP_END_OF_CYCLE : Bool;
         INMEDIATE_STOP : Bool;
         RESET_FAULTS : Bool;
      END_STRUCT;
      LAMPS : Struct
         CONTROL_ON : Bool;
         CONTROL_OFF : Bool;
         HOME_POSITION : Bool;
         AUTOMATIC_MODE : Bool;
         SEMIAUTOMATIC_MODE : Bool;
         MANUAL_MODE : Bool;
         START : Bool;
         STOP_END_OF_CYCLE : Bool;
         INMEDIATE_STOP : Bool;
         RESET_FAULTS : Bool;
      END_STRUCT;
   END_VAR
BEGIN
END_DATA_BLOCK

DATA_BLOCK "DB2000_WINCC_HMI_FUNCTION"   // DB2000
{ S7_Optimized_Access := 'FALSE'; DB_Accessible_From_OPC_UA := 'FALSE' }
AUTHOR : ETXETAR
VERSION : 1.0
// stored: AutoNumber false, DBAccessibleFromOPCUA false, DBAccessibleFromWebserver true, IsOnlyStoredInLoadMemory false, IsWriteProtectedInAS false
   VAR RETAIN
      HELP_PROMPT : Int;   // HELP PROMPT
      WINCC_SCREEN_NUMBER : Int;   // WINCC HMI SCREEN NUMBER
      PLC_SCREEN_SELECTION : Word;   // PLC SCREEN SELECTION
      SCREEN_SELECTION : Array[11..89] of Bool;   // SCREEN SELECTION
   END_VAR
BEGIN
END_DATA_BLOCK

